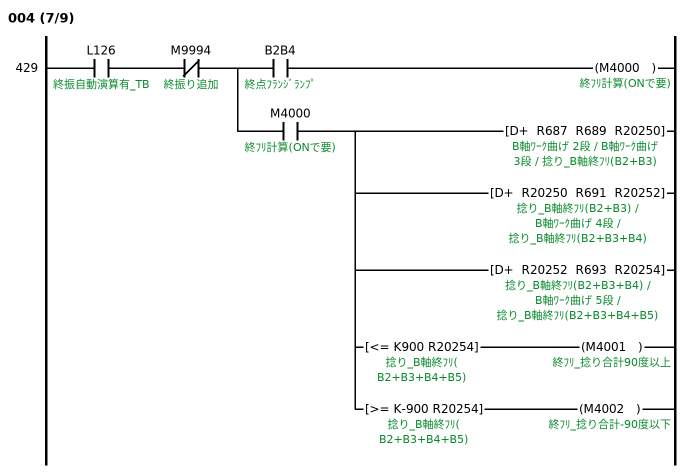
429   LD      L126  ; 終振自動演算有_TB
      ANI     M9994  ; 終振り追加
      MPS
      AND     B2B4  ; 終点ﾌﾗﾝｼﾞﾗﾝﾌﾟ
      OUT     M4000  ; 終ﾌﾘ計算(ONで要)
      MPP
      AND     M4000  ; 終ﾌﾘ計算(ONで要)
      D+      R687 R689 R20250  ; B軸ﾜｰｸ曲げ 2段 / B軸ﾜｰｸ曲げ 3段 / 捻り_B軸終ﾌﾘ(B2+B3)
      D+      R20250 R691 R20252  ; B軸ﾜｰｸ曲げ 4段 / 捻り_B軸終ﾌﾘ(B2+B3+B4)
      D+      R20252 R693 R20254  ; B軸ﾜｰｸ曲げ 5段 / 捻り_B軸終ﾌﾘ(B2+B3+B4+B5)
      MPS
      AND<=   K900 R20254  ; 捻り_B軸終ﾌﾘ(B2+B3+B4+B5)
      OUT     M4001  ; 終ﾌﾘ_捻り合計90度以上
      MPP
      AND>=   K-900 R20254  ; 捻り_B軸終ﾌﾘ(B2+B3+B4+B5)
      OUT     M4002  ; 終ﾌﾘ_捻り合計-90度以下
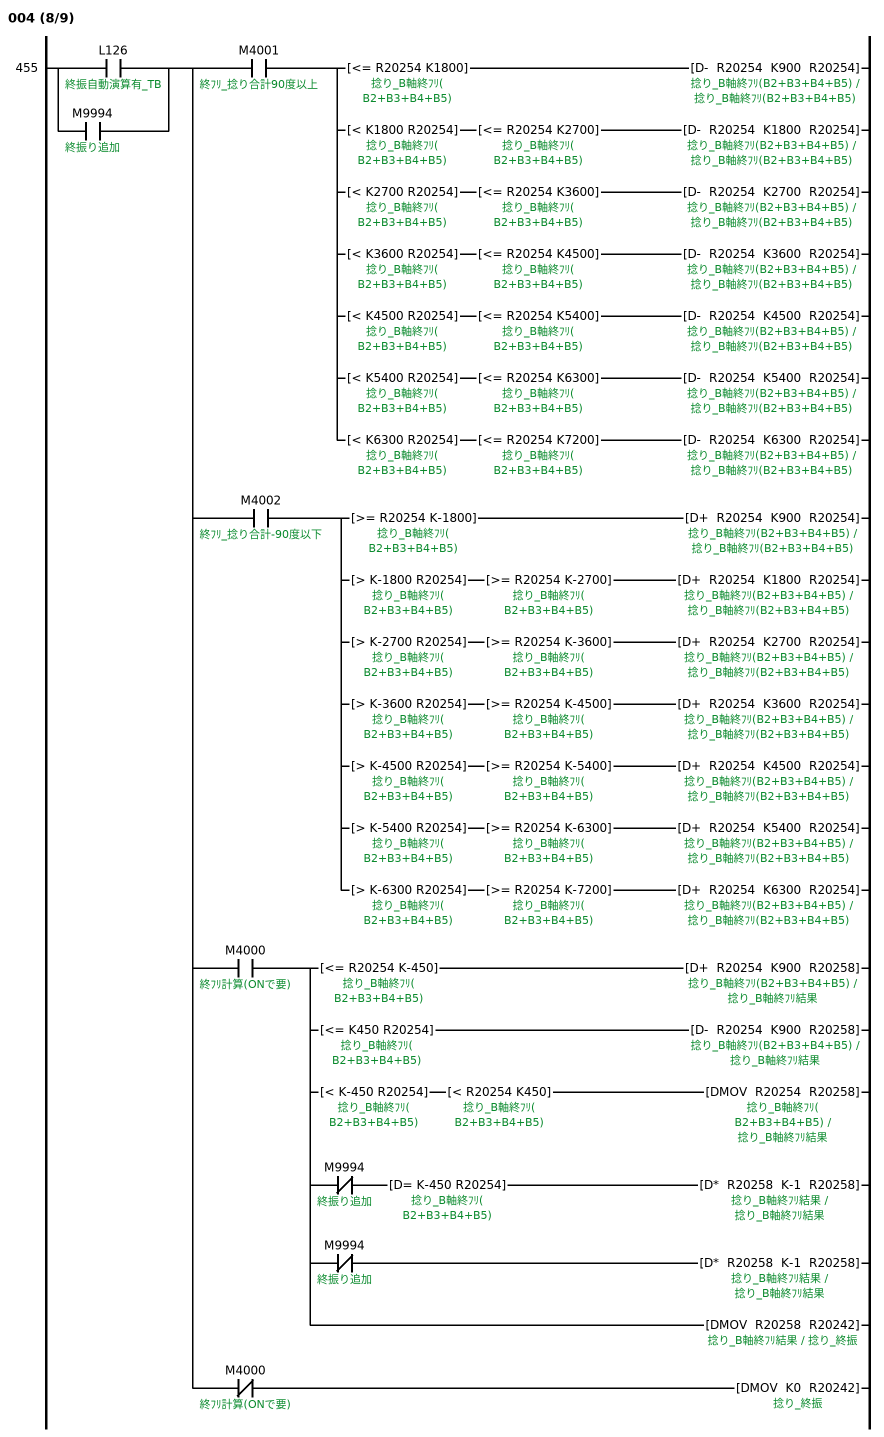
455   LD      L126  ; 終振自動演算有_TB
      OR      M9994  ; 終振り追加
      MPS
      AND     M4001  ; 終ﾌﾘ_捻り合計90度以上
      MPS
      AND<=   R20254 K1800  ; 捻り_B軸終ﾌﾘ(B2+B3+B4+B5)
      D-      R20254 K900 R20254
      MRD
      AND<    K1800 R20254  ; 捻り_B軸終ﾌﾘ(B2+B3+B4+B5)
      AND<=   R20254 K2700  ; 捻り_B軸終ﾌﾘ(B2+B3+B4+B5)
      D-      R20254 K1800 R20254
      MRD
      AND<    K2700 R20254  ; 捻り_B軸終ﾌﾘ(B2+B3+B4+B5)
      AND<=   R20254 K3600  ; 捻り_B軸終ﾌﾘ(B2+B3+B4+B5)
      D-      R20254 K2700 R20254
      MRD
      AND<    K3600 R20254  ; 捻り_B軸終ﾌﾘ(B2+B3+B4+B5)
      AND<=   R20254 K4500  ; 捻り_B軸終ﾌﾘ(B2+B3+B4+B5)
      D-      R20254 K3600 R20254
      MRD
      AND<    K4500 R20254  ; 捻り_B軸終ﾌﾘ(B2+B3+B4+B5)
      AND<=   R20254 K5400  ; 捻り_B軸終ﾌﾘ(B2+B3+B4+B5)
      D-      R20254 K4500 R20254
      MRD
      AND<    K5400 R20254  ; 捻り_B軸終ﾌﾘ(B2+B3+B4+B5)
      AND<=   R20254 K6300  ; 捻り_B軸終ﾌﾘ(B2+B3+B4+B5)
      D-      R20254 K5400 R20254
      MPP
      AND<    K6300 R20254  ; 捻り_B軸終ﾌﾘ(B2+B3+B4+B5)
      AND<=   R20254 K7200  ; 捻り_B軸終ﾌﾘ(B2+B3+B4+B5)
      D-      R20254 K6300 R20254
      MRD
      AND     M4002  ; 終ﾌﾘ_捻り合計-90度以下
      MPS
      AND>=   R20254 K-1800  ; 捻り_B軸終ﾌﾘ(B2+B3+B4+B5)
      D+      R20254 K900 R20254
      MRD
      AND>    K-1800 R20254  ; 捻り_B軸終ﾌﾘ(B2+B3+B4+B5)
      AND>=   R20254 K-2700  ; 捻り_B軸終ﾌﾘ(B2+B3+B4+B5)
      D+      R20254 K1800 R20254
      MRD
      AND>    K-2700 R20254  ; 捻り_B軸終ﾌﾘ(B2+B3+B4+B5)
      AND>=   R20254 K-3600  ; 捻り_B軸終ﾌﾘ(B2+B3+B4+B5)
      D+      R20254 K2700 R20254
      MRD
      AND>    K-3600 R20254  ; 捻り_B軸終ﾌﾘ(B2+B3+B4+B5)
      AND>=   R20254 K-4500  ; 捻り_B軸終ﾌﾘ(B2+B3+B4+B5)
      D+      R20254 K3600 R20254
      MRD
      AND>    K-4500 R20254  ; 捻り_B軸終ﾌﾘ(B2+B3+B4+B5)
      AND>=   R20254 K-5400  ; 捻り_B軸終ﾌﾘ(B2+B3+B4+B5)
      D+      R20254 K4500 R20254
      MRD
      AND>    K-5400 R20254  ; 捻り_B軸終ﾌﾘ(B2+B3+B4+B5)
      AND>=   R20254 K-6300  ; 捻り_B軸終ﾌﾘ(B2+B3+B4+B5)
      D+      R20254 K5400 R20254
      MPP
      AND>    K-6300 R20254  ; 捻り_B軸終ﾌﾘ(B2+B3+B4+B5)
      AND>=   R20254 K-7200  ; 捻り_B軸終ﾌﾘ(B2+B3+B4+B5)
      D+      R20254 K6300 R20254
      MRD
      AND     M4000  ; 終ﾌﾘ計算(ONで要)
      MPS
      AND<=   R20254 K-450  ; 捻り_B軸終ﾌﾘ(B2+B3+B4+B5)
      D+      R20254 K900 R20258  ; 捻り_B軸終ﾌﾘ結果
      MRD
      AND<=   K450 R20254  ; 捻り_B軸終ﾌﾘ(B2+B3+B4+B5)
      D-      R20254 K900 R20258
      MRD
      AND<    K-450 R20254  ; 捻り_B軸終ﾌﾘ(B2+B3+B4+B5)
      AND<    R20254 K450  ; 捻り_B軸終ﾌﾘ(B2+B3+B4+B5)
      DMOV    R20254 R20258
      MRD
      ANI     M9994  ; 終振り追加
      ANDD=   K-450 R20254  ; 捻り_B軸終ﾌﾘ(B2+B3+B4+B5)
      D*      R20258 K-1 R20258
      MRD
      ANI     M9994  ; 終振り追加
      D*      R20258 K-1 R20258
      MPP
      DMOV    R20258 R20242
      MPP
      ANI     M4000  ; 終ﾌﾘ計算(ONで要)
      DMOV    K0 R20242
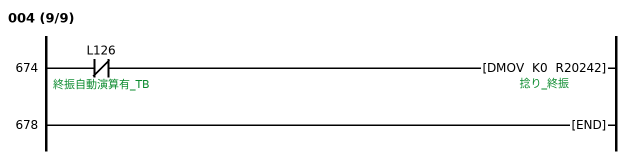
674   LDI     L126  ; 終振自動演算有_TB
      DMOV    K0 R20242
678   END
END_PROGRAM

PROGRAM 006  // 原点復帰
; 
      P600
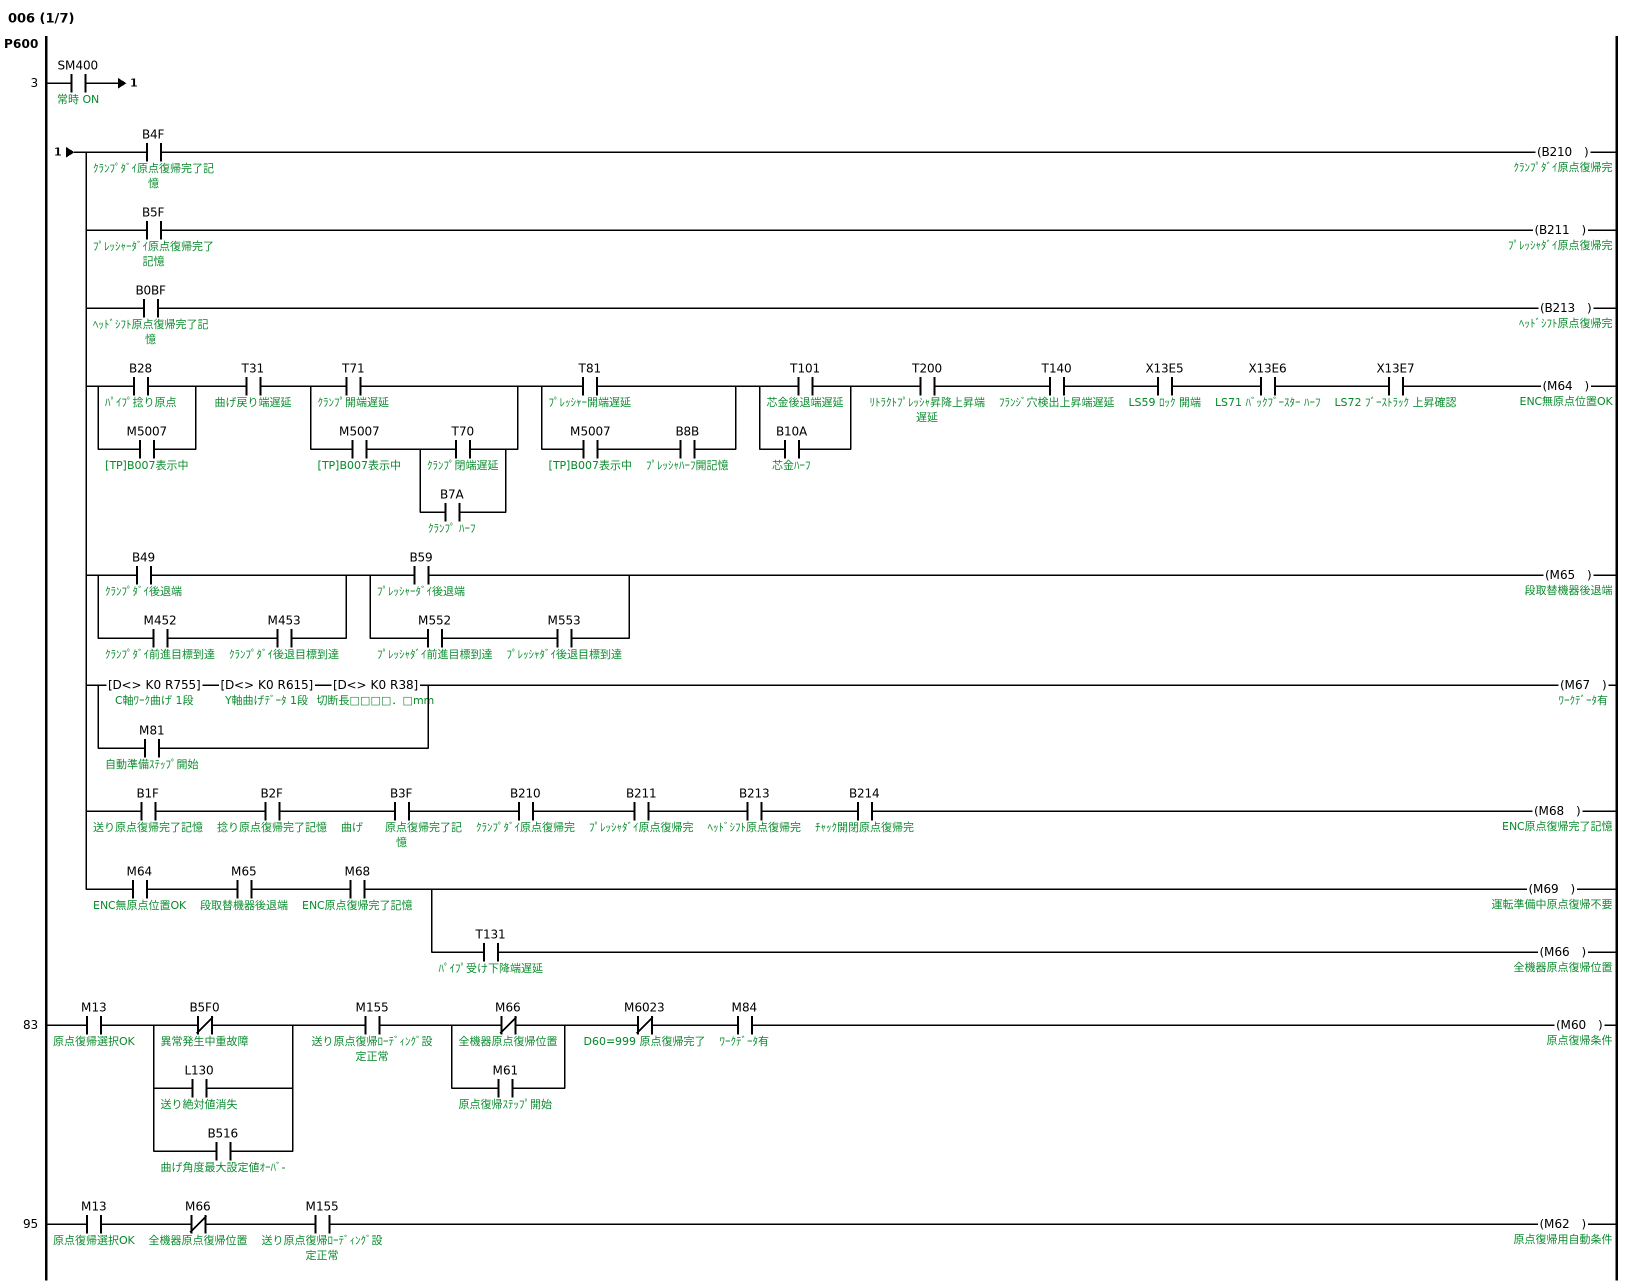
3     LD      SM400  ; 常時 ON
      MPS
      AND     B4F  ; ｸﾗﾝﾌﾟﾀﾞｲ原点復帰完了記憶
      OUT     B210  ; ｸﾗﾝﾌﾟﾀﾞｲ原点復帰完
      MRD
      AND     B5F  ; ﾌﾟﾚｯｼｬｰﾀﾞｲ原点復帰完了記憶
      OUT     B211  ; ﾌﾟﾚｯｼｬﾀﾞｲ原点復帰完
      MRD
      AND     B0BF  ; ﾍｯﾄﾞｼﾌﾄ原点復帰完了記憶
      OUT     B213  ; ﾍｯﾄﾞｼﾌﾄ原点復帰完
      MRD
      LD      B28  ; ﾊﾟｲﾌﾟ捻り原点
      OR      M5007  ; [TP]B007表示中
      ANB
      AND     T31  ; 曲げ戻り端遅延
      LD      T71  ; ｸﾗﾝﾌﾟ開端遅延
      LD      M5007  ; [TP]B007表示中
      LD      T70  ; ｸﾗﾝﾌﾟ閉端遅延
      OR      B7A  ; ｸﾗﾝﾌﾟ ﾊｰﾌ
      ANB
      ORB
      ANB
      LD      T81  ; ﾌﾟﾚｯｼｬｰ開端遅延
      LD      M5007  ; [TP]B007表示中
      AND     B8B  ; ﾌﾟﾚｯｼｬﾊｰﾌ開記憶
      ORB
      ANB
      LD      T101  ; 芯金後退端遅延
      OR      B10A  ; 芯金ﾊｰﾌ
      ANB
      AND     T200  ; ﾘﾄﾗｸﾄﾌﾟﾚｯｼｬ昇降上昇端遅延
      AND     T140  ; ﾌﾗﾝｼﾞ穴検出上昇端遅延
      AND     X13E5  ; LS59 ﾛｯｸ 開端
      AND     X13E6  ; LS71 ﾊﾞｯｸﾌﾞｰｽﾀｰ ﾊｰﾌ
      AND     X13E7  ; LS72 ﾌﾞｰｽﾄﾗｯｸ 上昇確認
      OUT     M64  ; ENC無原点位置OK
      MRD
      LD      B49  ; ｸﾗﾝﾌﾟﾀﾞｲ後退端
      LD      M452  ; ｸﾗﾝﾌﾟﾀﾞｲ前進目標到達
      AND     M453  ; ｸﾗﾝﾌﾟﾀﾞｲ後退目標到達
      ORB
      ANB
      LD      B59  ; ﾌﾟﾚｯｼｬｰﾀﾞｲ後退端
      LD      M552  ; ﾌﾟﾚｯｼｬﾀﾞｲ前進目標到達
      AND     M553  ; ﾌﾟﾚｯｼｬﾀﾞｲ後退目標到達
      ORB
      ANB
      OUT     M65  ; 段取替機器後退端
      MRD
      LDD<>   K0 R755  ; C軸ﾜｰｸ曲げ 1段
      ANDD<>  K0 R615  ; Y軸曲げﾃﾞｰﾀ 1段
      ANDD<>  K0 R38  ; 切断長□□□□．□mm
      OR      M81  ; 自動準備ｽﾃｯﾌﾟ開始
      ANB
      OUT     M67  ; ﾜｰｸﾃﾞｰﾀ有
      MRD
      AND     B1F  ; 送り原点復帰完了記憶
      AND     B2F  ; 捻り原点復帰完了記憶
      AND     B3F  ; 曲げ　　原点復帰完了記憶
      AND     B210  ; ｸﾗﾝﾌﾟﾀﾞｲ原点復帰完
      AND     B211  ; ﾌﾟﾚｯｼｬﾀﾞｲ原点復帰完
      AND     B213  ; ﾍｯﾄﾞｼﾌﾄ原点復帰完
      AND     B214  ; ﾁｬｯｸ開閉原点復帰完
      OUT     M68  ; ENC原点復帰完了記憶
      MPP
      AND     M64  ; ENC無原点位置OK
      AND     M65  ; 段取替機器後退端
      AND     M68  ; ENC原点復帰完了記憶
      OUT     M69  ; 運転準備中原点復帰不要
      AND     T131  ; ﾊﾟｲﾌﾟ受け下降端遅延
      OUT     M66  ; 全機器原点復帰位置
83    LD      M13  ; 原点復帰選択OK
      LDI     B5F0  ; 異常発生中重故障
      OR      L130  ; 送り絶対値消失
      OR      B516  ; 曲げ角度最大設定値ｵｰﾊﾞ-
      ANB
      AND     M155  ; 送り原点復帰ﾛｰﾃﾞｨﾝｸﾞ設定正常
      LDI     M66  ; 全機器原点復帰位置
      OR      M61  ; 原点復帰ｽﾃｯﾌﾟ開始
      ANB
      ANI     M6023  ; D60=999 原点復帰完了
      AND     M84  ; ﾜｰｸﾃﾞｰﾀ有
      OUT     M60  ; 原点復帰条件
95    LD      M13  ; 原点復帰選択OK
      ANI     M66  ; 全機器原点復帰位置
      AND     M155  ; 送り原点復帰ﾛｰﾃﾞｨﾝｸﾞ設定正常
      OUT     M62  ; 原点復帰用自動条件
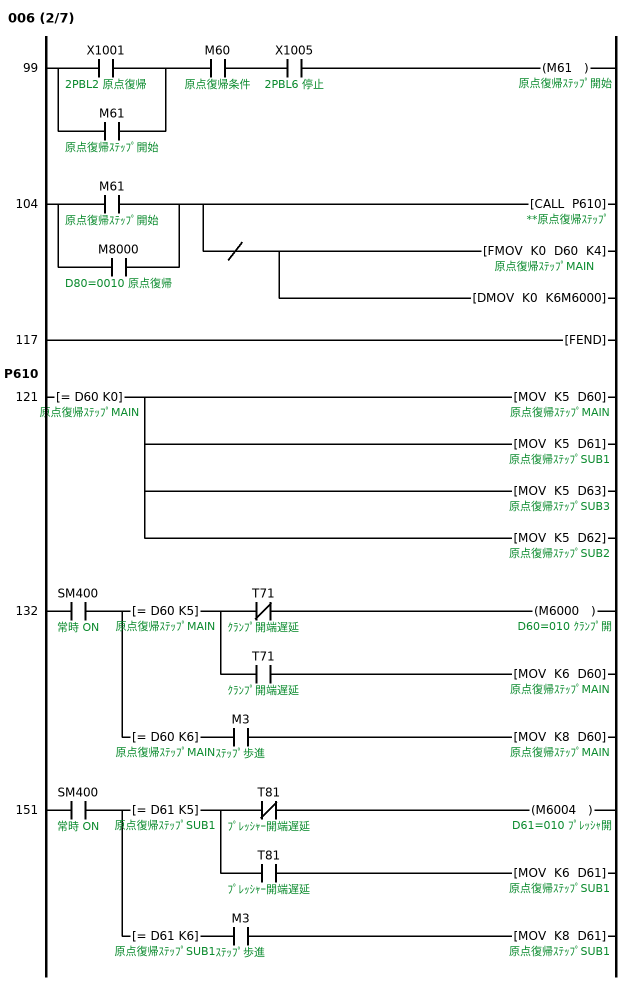
99    LD      X1001  ; 2PBL2 原点復帰
      OR      M61  ; 原点復帰ｽﾃｯﾌﾟ開始
      AND     M60  ; 原点復帰条件
      AND     X1005  ; 2PBL6 停止
      OUT     M61  ; 原点復帰ｽﾃｯﾌﾟ開始
104   LD      M61  ; 原点復帰ｽﾃｯﾌﾟ開始
      OR      M8000  ; D80=0010 原点復帰
      CALL    P610  ; **原点復帰ｽﾃｯﾌﾟ
      INV
      FMOV    K0 D60 K4  ; 原点復帰ｽﾃｯﾌﾟMAIN
      DMOV    K0 K6M6000  ; D60=010 ｸﾗﾝﾌﾟ開
117   FEND
; 
      P610
121   LD=     D60 K0  ; 原点復帰ｽﾃｯﾌﾟMAIN
      MOV     K5 D60
      MOV     K5 D61  ; 原点復帰ｽﾃｯﾌﾟSUB1
      MOV     K5 D63  ; 原点復帰ｽﾃｯﾌﾟSUB3
      MOV     K5 D62  ; 原点復帰ｽﾃｯﾌﾟSUB2
132   LD      SM400  ; 常時 ON
      MPS
      AND=    D60 K5  ; 原点復帰ｽﾃｯﾌﾟMAIN
      MPS
      ANI     T71  ; ｸﾗﾝﾌﾟ開端遅延
      OUT     M6000  ; D60=010 ｸﾗﾝﾌﾟ開
      MPP
      AND     T71  ; ｸﾗﾝﾌﾟ開端遅延
      MOV     K6 D60
      MPP
      AND=    D60 K6  ; 原点復帰ｽﾃｯﾌﾟMAIN
      AND     M3  ; ｽﾃｯﾌﾟ歩進
      MOV     K8 D60
151   LD      SM400  ; 常時 ON
      MPS
      AND=    D61 K5  ; 原点復帰ｽﾃｯﾌﾟSUB1
      MPS
      ANI     T81  ; ﾌﾟﾚｯｼｬｰ開端遅延
      OUT     M6004  ; D61=010 ﾌﾟﾚｯｼｬ開
      MPP
      AND     T81  ; ﾌﾟﾚｯｼｬｰ開端遅延
      MOV     K6 D61
      MPP
      AND=    D61 K6  ; 原点復帰ｽﾃｯﾌﾟSUB1
      AND     M3  ; ｽﾃｯﾌﾟ歩進
      MOV     K8 D61
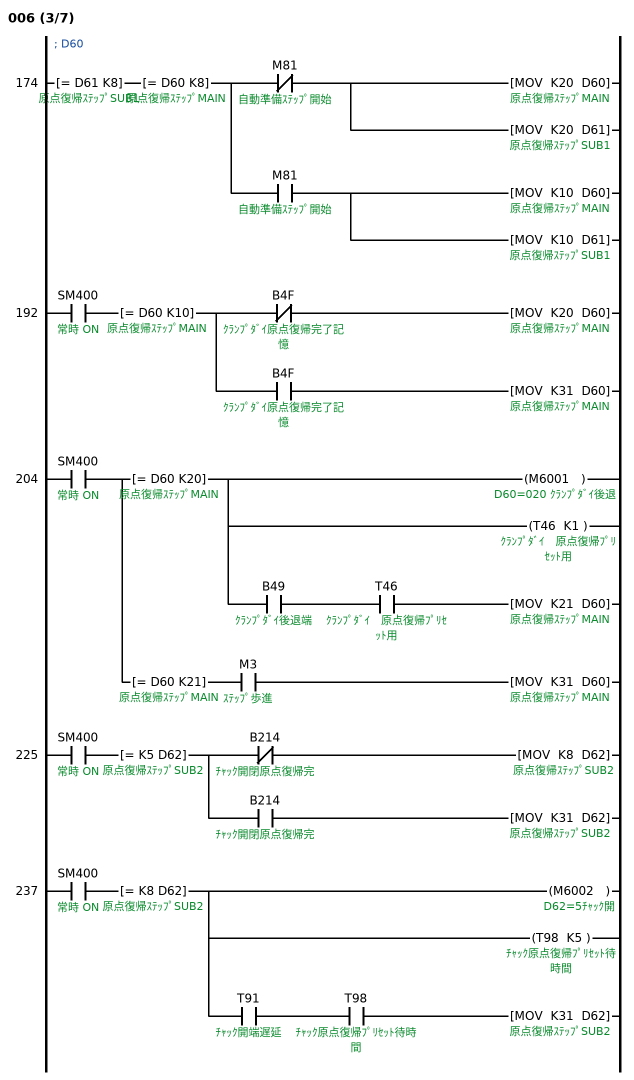
; D60
174   LD=     D61 K8  ; 原点復帰ｽﾃｯﾌﾟSUB1
      AND=    D60 K8  ; 原点復帰ｽﾃｯﾌﾟMAIN
      MPS
      ANI     M81  ; 自動準備ｽﾃｯﾌﾟ開始
      MOV     K20 D60
      MOV     K20 D61
      MPP
      AND     M81  ; 自動準備ｽﾃｯﾌﾟ開始
      MOV     K10 D60
      MOV     K10 D61
192   LD      SM400  ; 常時 ON
      AND=    D60 K10  ; 原点復帰ｽﾃｯﾌﾟMAIN
      MPS
      ANI     B4F  ; ｸﾗﾝﾌﾟﾀﾞｲ原点復帰完了記憶
      MOV     K20 D60
      MPP
      AND     B4F  ; ｸﾗﾝﾌﾟﾀﾞｲ原点復帰完了記憶
      MOV     K31 D60
204   LD      SM400  ; 常時 ON
      MPS
      AND=    D60 K20  ; 原点復帰ｽﾃｯﾌﾟMAIN
      OUT     M6001  ; D60=020 ｸﾗﾝﾌﾟﾀﾞｲ後退
      OUT     T46 K1  ; ｸﾗﾝﾌﾟﾀﾞｲ　原点復帰ﾌﾟﾘｾｯﾄ用
      AND     B49  ; ｸﾗﾝﾌﾟﾀﾞｲ後退端
      AND     T46  ; ｸﾗﾝﾌﾟﾀﾞｲ　原点復帰ﾌﾟﾘｾｯﾄ用
      MOV     K21 D60
      MPP
      AND=    D60 K21  ; 原点復帰ｽﾃｯﾌﾟMAIN
      AND     M3  ; ｽﾃｯﾌﾟ歩進
      MOV     K31 D60
225   LD      SM400  ; 常時 ON
      AND=    K5 D62  ; 原点復帰ｽﾃｯﾌﾟSUB2
      MPS
      ANI     B214  ; ﾁｬｯｸ開閉原点復帰完
      MOV     K8 D62
      MPP
      AND     B214  ; ﾁｬｯｸ開閉原点復帰完
      MOV     K31 D62
237   LD      SM400  ; 常時 ON
      AND=    K8 D62  ; 原点復帰ｽﾃｯﾌﾟSUB2
      OUT     M6002  ; D62=5ﾁｬｯｸ開
      OUT     T98 K5  ; ﾁｬｯｸ原点復帰ﾌﾟﾘｾｯﾄ待時間
      AND     T91  ; ﾁｬｯｸ開端遅延
      AND     T98  ; ﾁｬｯｸ原点復帰ﾌﾟﾘｾｯﾄ待時間
      MOV     K31 D62
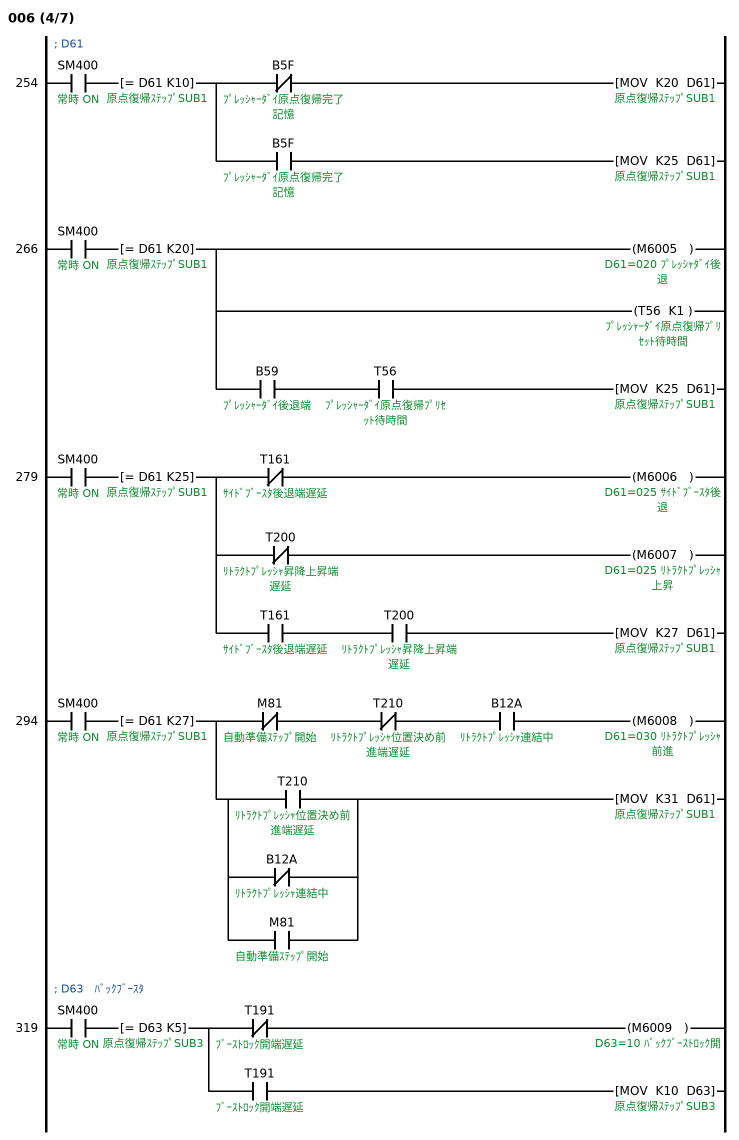
; D61
254   LD      SM400  ; 常時 ON
      AND=    D61 K10  ; 原点復帰ｽﾃｯﾌﾟSUB1
      MPS
      ANI     B5F  ; ﾌﾟﾚｯｼｬｰﾀﾞｲ原点復帰完了記憶
      MOV     K20 D61
      MPP
      AND     B5F  ; ﾌﾟﾚｯｼｬｰﾀﾞｲ原点復帰完了記憶
      MOV     K25 D61
266   LD      SM400  ; 常時 ON
      AND=    D61 K20  ; 原点復帰ｽﾃｯﾌﾟSUB1
      OUT     M6005  ; D61=020 ﾌﾟﾚｯｼｬﾀﾞｲ後退
      OUT     T56 K1  ; ﾌﾟﾚｯｼｬｰﾀﾞｲ原点復帰ﾌﾟﾘｾｯﾄ待時間
      AND     B59  ; ﾌﾟﾚｯｼｬｰﾀﾞｲ後退端
      AND     T56  ; ﾌﾟﾚｯｼｬｰﾀﾞｲ原点復帰ﾌﾟﾘｾｯﾄ待時間
      MOV     K25 D61
279   LD      SM400  ; 常時 ON
      AND=    D61 K25  ; 原点復帰ｽﾃｯﾌﾟSUB1
      MPS
      ANI     T161  ; ｻｲﾄﾞﾌﾞｰｽﾀ後退端遅延
      OUT     M6006  ; D61=025 ｻｲﾄﾞﾌﾞｰｽﾀ後退
      MRD
      ANI     T200  ; ﾘﾄﾗｸﾄﾌﾟﾚｯｼｬ昇降上昇端遅延
      OUT     M6007  ; D61=025 ﾘﾄﾗｸﾄﾌﾟﾚｯｼｬ上昇
      MPP
      AND     T161  ; ｻｲﾄﾞﾌﾞｰｽﾀ後退端遅延
      AND     T200  ; ﾘﾄﾗｸﾄﾌﾟﾚｯｼｬ昇降上昇端遅延
      MOV     K27 D61
294   LD      SM400  ; 常時 ON
      AND=    D61 K27  ; 原点復帰ｽﾃｯﾌﾟSUB1
      MPS
      ANI     M81  ; 自動準備ｽﾃｯﾌﾟ開始
      ANI     T210  ; ﾘﾄﾗｸﾄﾌﾟﾚｯｼｬ位置決め前進端遅延
      AND     B12A  ; ﾘﾄﾗｸﾄﾌﾟﾚｯｼｬ連結中
      OUT     M6008  ; D61=030 ﾘﾄﾗｸﾄﾌﾟﾚｯｼｬ前進
      MPP
      LD      T210  ; ﾘﾄﾗｸﾄﾌﾟﾚｯｼｬ位置決め前進端遅延
      ORI     B12A  ; ﾘﾄﾗｸﾄﾌﾟﾚｯｼｬ連結中
      OR      M81  ; 自動準備ｽﾃｯﾌﾟ開始
      ANB
      MOV     K31 D61
; D63　ﾊﾞｯｸﾌﾞｰｽﾀ
319   LD      SM400  ; 常時 ON
      AND=    D63 K5  ; 原点復帰ｽﾃｯﾌﾟSUB3
      MPS
      ANI     T191  ; ﾌﾞｰｽﾄﾛｯｸ開端遅延
      OUT     M6009  ; D63=10 ﾊﾞｯｸﾌﾞｰｽﾄﾛｯｸ開
      MPP
      AND     T191  ; ﾌﾞｰｽﾄﾛｯｸ開端遅延
      MOV     K10 D63
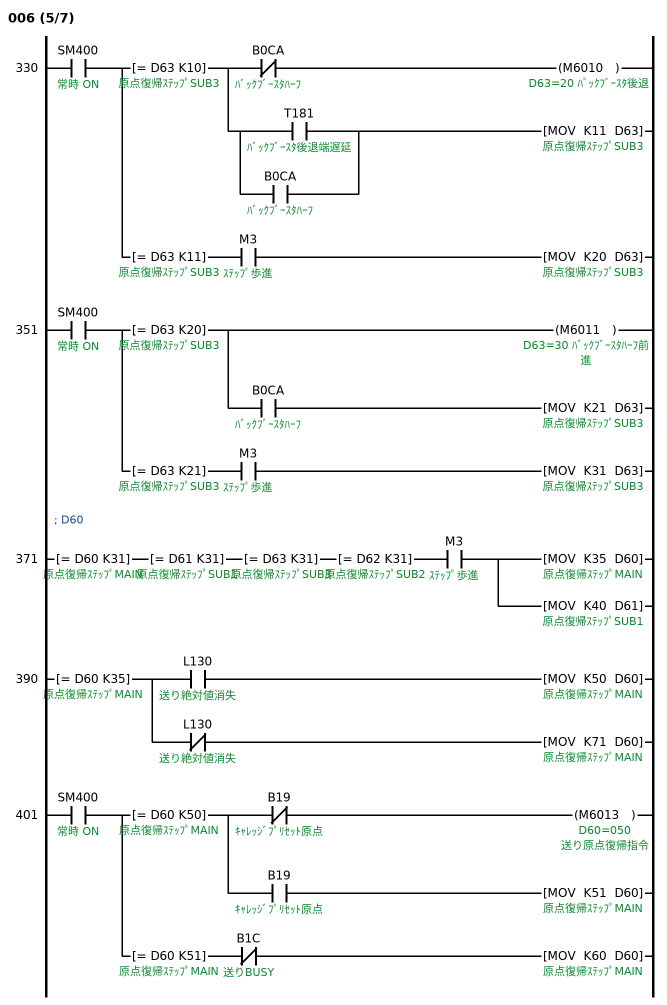
330   LD      SM400  ; 常時 ON
      MPS
      AND=    D63 K10  ; 原点復帰ｽﾃｯﾌﾟSUB3
      MPS
      ANI     B0CA  ; ﾊﾞｯｸﾌﾞｰｽﾀﾊｰﾌ
      OUT     M6010  ; D63=20 ﾊﾞｯｸﾌﾞｰｽﾀ後退
      MPP
      LD      T181  ; ﾊﾞｯｸﾌﾞｰｽﾀ後退端遅延
      OR      B0CA  ; ﾊﾞｯｸﾌﾞｰｽﾀﾊｰﾌ
      ANB
      MOV     K11 D63
      MPP
      AND=    D63 K11  ; 原点復帰ｽﾃｯﾌﾟSUB3
      AND     M3  ; ｽﾃｯﾌﾟ歩進
      MOV     K20 D63
351   LD      SM400  ; 常時 ON
      MPS
      AND=    D63 K20  ; 原点復帰ｽﾃｯﾌﾟSUB3
      OUT     M6011  ; D63=30 ﾊﾞｯｸﾌﾞｰｽﾀﾊｰﾌ前進
      AND     B0CA  ; ﾊﾞｯｸﾌﾞｰｽﾀﾊｰﾌ
      MOV     K21 D63
      MPP
      AND=    D63 K21  ; 原点復帰ｽﾃｯﾌﾟSUB3
      AND     M3  ; ｽﾃｯﾌﾟ歩進
      MOV     K31 D63
; D60
371   LD=     D60 K31  ; 原点復帰ｽﾃｯﾌﾟMAIN
      AND=    D61 K31  ; 原点復帰ｽﾃｯﾌﾟSUB1
      AND=    D63 K31  ; 原点復帰ｽﾃｯﾌﾟSUB3
      AND=    D62 K31  ; 原点復帰ｽﾃｯﾌﾟSUB2
      AND     M3  ; ｽﾃｯﾌﾟ歩進
      MOV     K35 D60
      MOV     K40 D61
; 
390   LD=     D60 K35  ; 原点復帰ｽﾃｯﾌﾟMAIN
      MPS
      AND     L130  ; 送り絶対値消失
      MOV     K50 D60
      MPP
      ANI     L130  ; 送り絶対値消失
      MOV     K71 D60
401   LD      SM400  ; 常時 ON
      MPS
      AND=    D60 K50  ; 原点復帰ｽﾃｯﾌﾟMAIN
      MPS
      ANI     B19  ; ｷｬﾚｯｼﾞﾌﾟﾘｾｯﾄ原点
      OUT     M6013  ; D60=050 送り原点復帰指令
      MPP
      AND     B19  ; ｷｬﾚｯｼﾞﾌﾟﾘｾｯﾄ原点
      MOV     K51 D60
      MPP
      AND=    D60 K51  ; 原点復帰ｽﾃｯﾌﾟMAIN
      ANI     B1C  ; 送りBUSY
      MOV     K60 D60
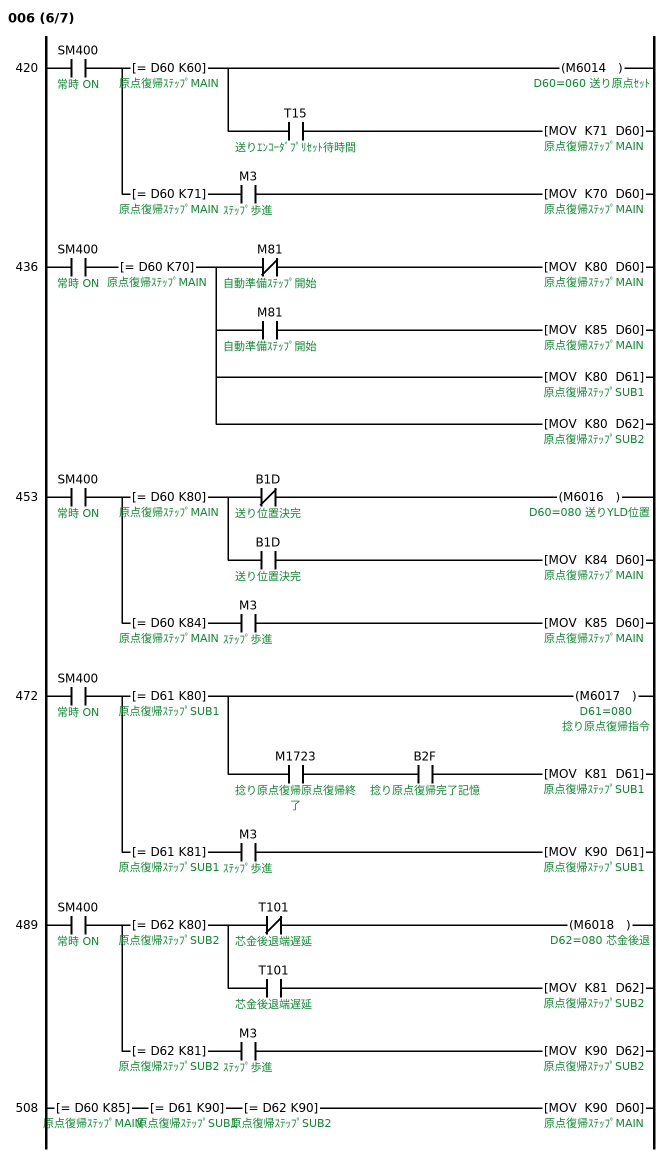
420   LD      SM400  ; 常時 ON
      MPS
      AND=    D60 K60  ; 原点復帰ｽﾃｯﾌﾟMAIN
      OUT     M6014  ; D60=060 送り原点ｾｯﾄ
      AND     T15  ; 送りｴﾝｺｰﾀﾞﾌﾟﾘｾｯﾄ待時間
      MOV     K71 D60
      MPP
      AND=    D60 K71  ; 原点復帰ｽﾃｯﾌﾟMAIN
      AND     M3  ; ｽﾃｯﾌﾟ歩進
      MOV     K70 D60
436   LD      SM400  ; 常時 ON
      AND=    D60 K70  ; 原点復帰ｽﾃｯﾌﾟMAIN
      MPS
      ANI     M81  ; 自動準備ｽﾃｯﾌﾟ開始
      MOV     K80 D60
      MRD
      AND     M81  ; 自動準備ｽﾃｯﾌﾟ開始
      MOV     K85 D60
      MPP
      MOV     K80 D61
      MOV     K80 D62
453   LD      SM400  ; 常時 ON
      MPS
      AND=    D60 K80  ; 原点復帰ｽﾃｯﾌﾟMAIN
      MPS
      ANI     B1D  ; 送り位置決完
      OUT     M6016  ; D60=080 送りYLD位置
      MPP
      AND     B1D  ; 送り位置決完
      MOV     K84 D60
      MPP
      AND=    D60 K84  ; 原点復帰ｽﾃｯﾌﾟMAIN
      AND     M3  ; ｽﾃｯﾌﾟ歩進
      MOV     K85 D60
472   LD      SM400  ; 常時 ON
      MPS
      AND=    D61 K80  ; 原点復帰ｽﾃｯﾌﾟSUB1
      OUT     M6017  ; D61=080 捻り原点復帰指令
      AND     M1723  ; 捻り原点復帰原点復帰終了
      AND     B2F  ; 捻り原点復帰完了記憶
      MOV     K81 D61
      MPP
      AND=    D61 K81  ; 原点復帰ｽﾃｯﾌﾟSUB1
      AND     M3  ; ｽﾃｯﾌﾟ歩進
      MOV     K90 D61
489   LD      SM400  ; 常時 ON
      MPS
      AND=    D62 K80  ; 原点復帰ｽﾃｯﾌﾟSUB2
      MPS
      ANI     T101  ; 芯金後退端遅延
      OUT     M6018  ; D62=080 芯金後退
      MPP
      AND     T101  ; 芯金後退端遅延
      MOV     K81 D62
      MPP
      AND=    D62 K81  ; 原点復帰ｽﾃｯﾌﾟSUB2
      AND     M3  ; ｽﾃｯﾌﾟ歩進
      MOV     K90 D62
508   LD=     D60 K85  ; 原点復帰ｽﾃｯﾌﾟMAIN
      AND=    D61 K90  ; 原点復帰ｽﾃｯﾌﾟSUB1
      AND=    D62 K90  ; 原点復帰ｽﾃｯﾌﾟSUB2
      MOV     K90 D60
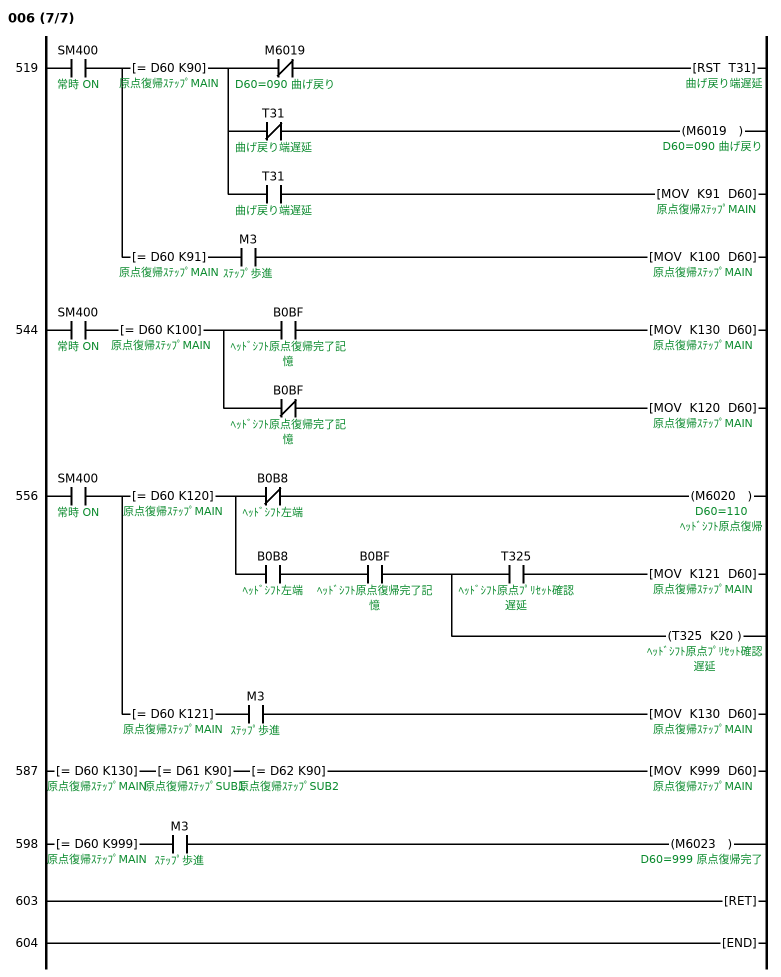
519   LD      SM400  ; 常時 ON
      MPS
      AND=    D60 K90  ; 原点復帰ｽﾃｯﾌﾟMAIN
      MPS
      ANI     M6019  ; D60=090 曲げ戻り
      RST     T31  ; 曲げ戻り端遅延
      MRD
      ANI     T31  ; 曲げ戻り端遅延
      OUT     M6019  ; D60=090 曲げ戻り
      MPP
      AND     T31  ; 曲げ戻り端遅延
      MOV     K91 D60
      MPP
      AND=    D60 K91  ; 原点復帰ｽﾃｯﾌﾟMAIN
      AND     M3  ; ｽﾃｯﾌﾟ歩進
      MOV     K100 D60
544   LD      SM400  ; 常時 ON
      AND=    D60 K100  ; 原点復帰ｽﾃｯﾌﾟMAIN
      MPS
      AND     B0BF  ; ﾍｯﾄﾞｼﾌﾄ原点復帰完了記憶
      MOV     K130 D60
      MPP
      ANI     B0BF  ; ﾍｯﾄﾞｼﾌﾄ原点復帰完了記憶
      MOV     K120 D60
556   LD      SM400  ; 常時 ON
      MPS
      AND=    D60 K120  ; 原点復帰ｽﾃｯﾌﾟMAIN
      MPS
      ANI     B0B8  ; ﾍｯﾄﾞｼﾌﾄ左端
      OUT     M6020  ; D60=110 ﾍｯﾄﾞｼﾌﾄ原点復帰
      MPP
      AND     B0B8  ; ﾍｯﾄﾞｼﾌﾄ左端
      AND     B0BF  ; ﾍｯﾄﾞｼﾌﾄ原点復帰完了記憶
      MPS
      AND     T325  ; ﾍｯﾄﾞｼﾌﾄ原点ﾌﾟﾘｾｯﾄ確認遅延
      MOV     K121 D60
      MPP
      OUT     T325 K20  ; ﾍｯﾄﾞｼﾌﾄ原点ﾌﾟﾘｾｯﾄ確認遅延
      MPP
      AND=    D60 K121  ; 原点復帰ｽﾃｯﾌﾟMAIN
      AND     M3  ; ｽﾃｯﾌﾟ歩進
      MOV     K130 D60
; 
; 
587   LD=     D60 K130  ; 原点復帰ｽﾃｯﾌﾟMAIN
      AND=    D61 K90  ; 原点復帰ｽﾃｯﾌﾟSUB1
      AND=    D62 K90  ; 原点復帰ｽﾃｯﾌﾟSUB2
      MOV     K999 D60
598   LD=     D60 K999  ; 原点復帰ｽﾃｯﾌﾟMAIN
      AND     M3  ; ｽﾃｯﾌﾟ歩進
      OUT     M6023  ; D60=999 原点復帰完了
603   RET
604   END
END_PROGRAM

PROGRAM 007  // 自動
; 
      P700
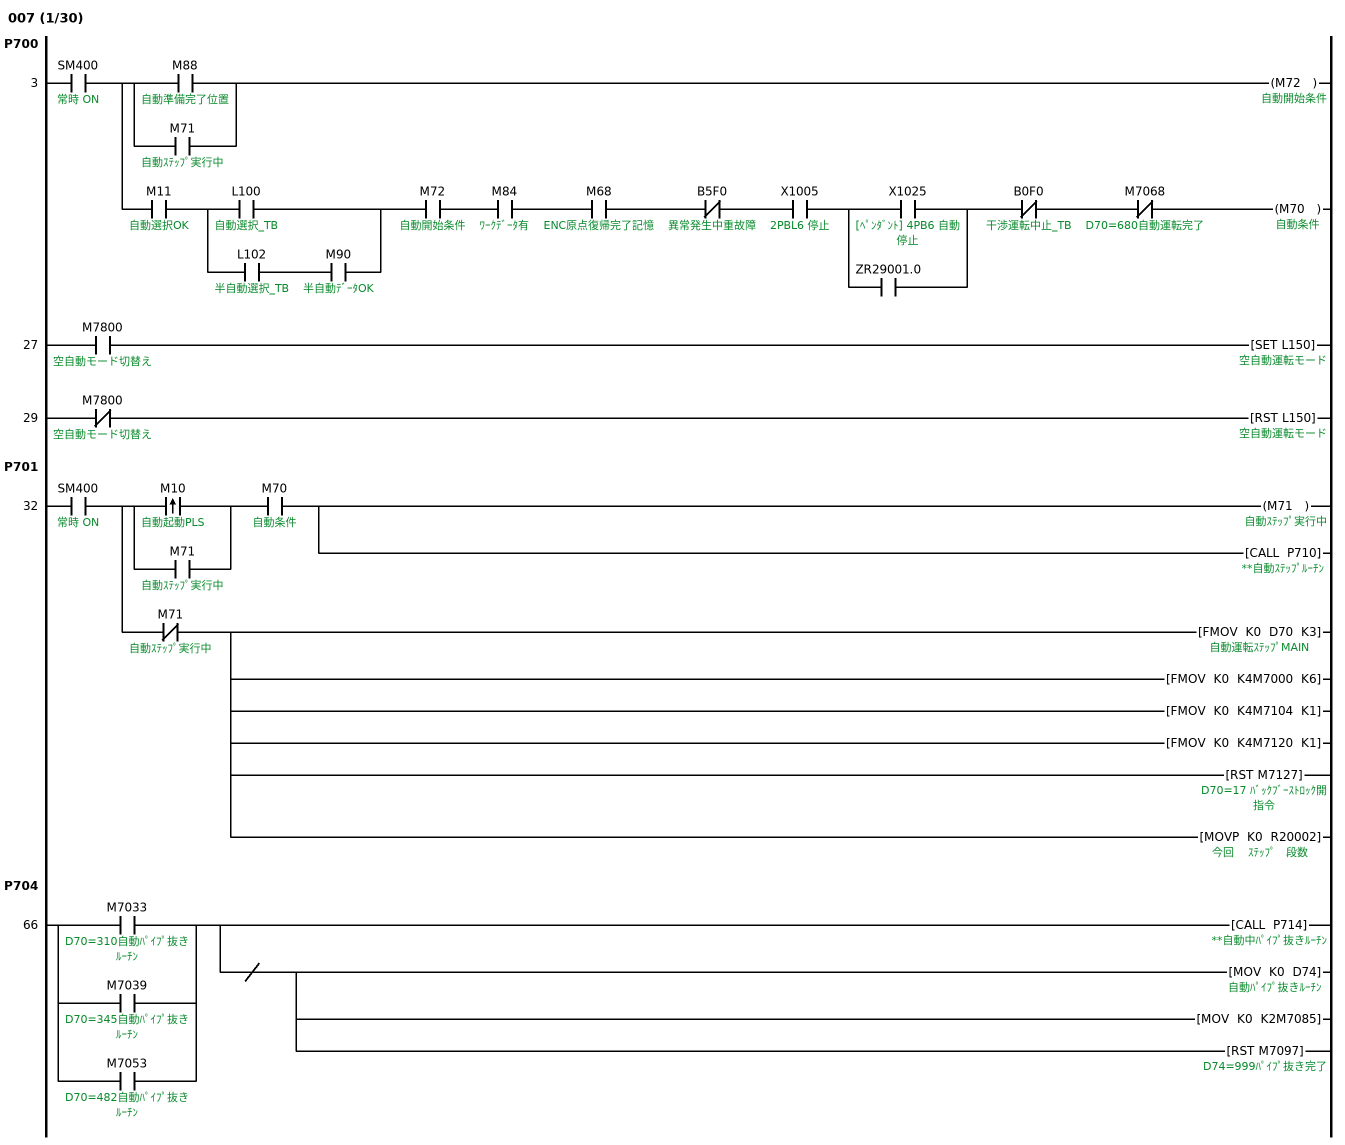
3     LD      SM400  ; 常時 ON
      MPS
      LD      M88  ; 自動準備完了位置
      OR      M71  ; 自動ｽﾃｯﾌﾟ実行中
      ANB
      OUT     M72  ; 自動開始条件
      MPP
      AND     M11  ; 自動選択OK
      LD      L100  ; 自動選択_TB
      LD      L102  ; 半自動選択_TB
      AND     M90  ; 半自動ﾃﾞｰﾀOK
      ORB
      ANB
      AND     M72  ; 自動開始条件
      AND     M84  ; ﾜｰｸﾃﾞｰﾀ有
      AND     M68  ; ENC原点復帰完了記憶
      ANI     B5F0  ; 異常発生中重故障
      AND     X1005  ; 2PBL6 停止
      LD      X1025  ; [ﾍﾟﾝﾀﾞﾝﾄ] 4PB6 自動 停止
      OR      ZR29001.0
      ANB
      ANI     B0F0  ; 干渉運転中止_TB
      ANI     M7068  ; D70=680自動運転完了
      OUT     M70  ; 自動条件
27    LD      M7800  ; 空自動モード切替え
      SET     L150  ; 空自動運転モード
29    LDI     M7800  ; 空自動モード切替え
      RST     L150  ; 空自動運転モード
      P701
32    LD      SM400  ; 常時 ON
      MPS
      LDP     M10  ; 自動起動PLS
      OR      M71  ; 自動ｽﾃｯﾌﾟ実行中
      ANB
      AND     M70  ; 自動条件
      OUT     M71  ; 自動ｽﾃｯﾌﾟ実行中
      CALL    P710  ; **自動ｽﾃｯﾌﾟﾙｰﾁﾝ
      MPP
      ANI     M71  ; 自動ｽﾃｯﾌﾟ実行中
      FMOV    K0 D70 K3  ; 自動運転ｽﾃｯﾌﾟMAIN
      FMOV    K0 K4M7000 K6  ; D70=000ﾃﾞｰﾀ確認
      FMOV    K0 K4M7104 K1  ; D70=590選択ﾛｯﾄ完了
      FMOV    K0 K4M7120 K1  ; D70=307ﾍｯﾄﾞｼﾌﾄ曲げ位置
      RST     M7127  ; D70=17 ﾊﾞｯｸﾌﾞｰｽﾄﾛｯｸ開指令
      MOVP    K0 R20002  ; 今回    ｽﾃｯﾌﾟ   段数
      P704
66    LD      M7033  ; D70=310自動ﾊﾟｲﾌﾟ抜きﾙｰﾁﾝ
      OR      M7039  ; D70=345自動ﾊﾟｲﾌﾟ抜きﾙｰﾁﾝ
      OR      M7053  ; D70=482自動ﾊﾟｲﾌﾟ抜きﾙｰﾁﾝ
      CALL    P714  ; **自動中ﾊﾟｲﾌﾟ抜きﾙｰﾁﾝ
      INV
      MOV     K0 D74  ; 自動ﾊﾟｲﾌﾟ抜きﾙｰﾁﾝ
      MOV     K0 K2M7085  ; D74=000予備
      RST     M7097  ; D74=999ﾊﾟｲﾌﾟ抜き完了
      P705
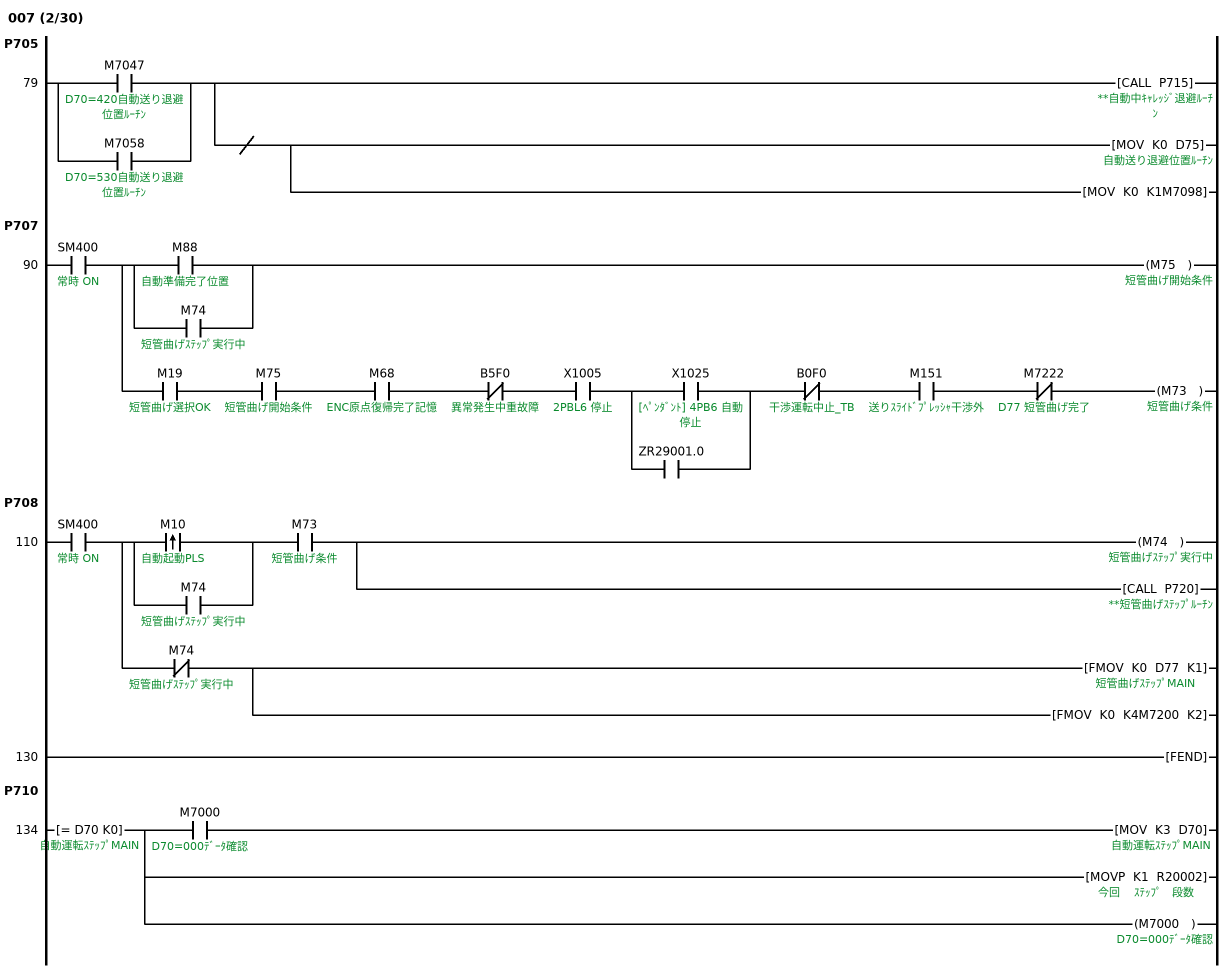
79    LD      M7047  ; D70=420自動送り退避位置ﾙｰﾁﾝ
      OR      M7058  ; D70=530自動送り退避位置ﾙｰﾁﾝ
      CALL    P715  ; **自動中ｷｬﾚｯｼﾞ退避ﾙｰﾁﾝ
      INV
      MOV     K0 D75  ; 自動送り退避位置ﾙｰﾁﾝ
      MOV     K0 K1M7098  ; D75=010送り退避位置
      P707
90    LD      SM400  ; 常時 ON
      MPS
      LD      M88  ; 自動準備完了位置
      OR      M74  ; 短管曲げｽﾃｯﾌﾟ実行中
      ANB
      OUT     M75  ; 短管曲げ開始条件
      MPP
      AND     M19  ; 短管曲げ選択OK
      AND     M75  ; 短管曲げ開始条件
      AND     M68  ; ENC原点復帰完了記憶
      ANI     B5F0  ; 異常発生中重故障
      AND     X1005  ; 2PBL6 停止
      LD      X1025  ; [ﾍﾟﾝﾀﾞﾝﾄ] 4PB6 自動 停止
      OR      ZR29001.0
      ANB
      ANI     B0F0  ; 干渉運転中止_TB
      AND     M151  ; 送りｽﾗｲﾄﾞﾌﾟﾚｯｼｬ干渉外
      ANI     M7222  ; D77 短管曲げ完了
      OUT     M73  ; 短管曲げ条件
      P708
110   LD      SM400  ; 常時 ON
      MPS
      LDP     M10  ; 自動起動PLS
      OR      M74  ; 短管曲げｽﾃｯﾌﾟ実行中
      ANB
      AND     M73  ; 短管曲げ条件
      OUT     M74  ; 短管曲げｽﾃｯﾌﾟ実行中
      CALL    P720  ; **短管曲げｽﾃｯﾌﾟﾙｰﾁﾝ
      MPP
      ANI     M74  ; 短管曲げｽﾃｯﾌﾟ実行中
      FMOV    K0 D77 K1  ; 短管曲げｽﾃｯﾌﾟMAIN
      FMOV    K0 K4M7200 K2
130   FEND
; 
      P710
134   LD=     D70 K0  ; 自動運転ｽﾃｯﾌﾟMAIN
      MPS
      AND     M7000  ; D70=000ﾃﾞｰﾀ確認
      MOV     K3 D70
      MPP
      MOVP    K1 R20002
      OUT     M7000  ; D70=000ﾃﾞｰﾀ確認
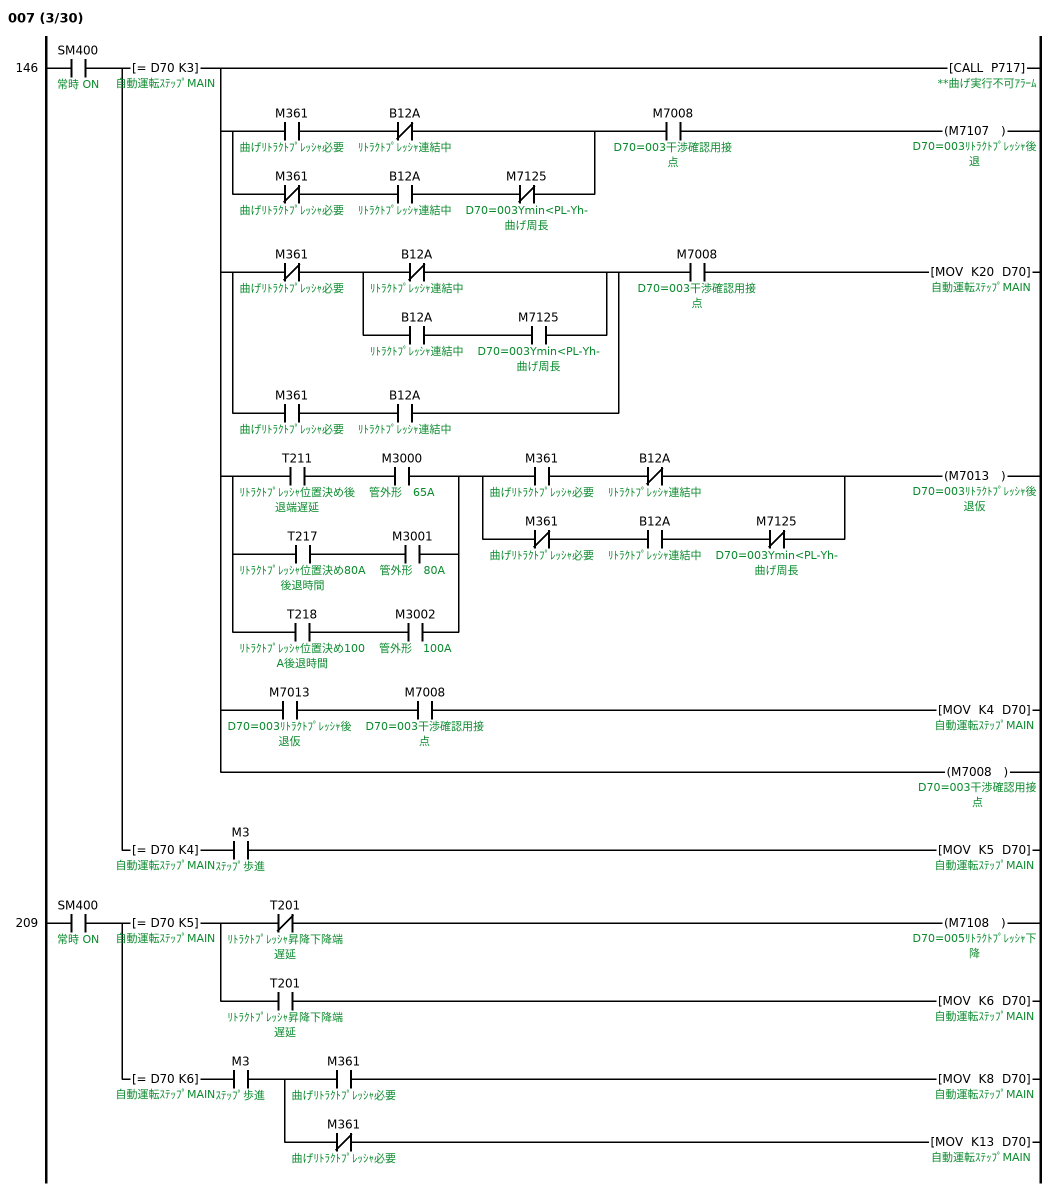
146   LD      SM400  ; 常時 ON
      MPS
      AND=    D70 K3  ; 自動運転ｽﾃｯﾌﾟMAIN
      CALL    P717  ; **曲げ実行不可ｱﾗｰﾑ
      MPS
      LD      M361  ; 曲げﾘﾄﾗｸﾄﾌﾟﾚｯｼｬ必要
      ANI     B12A  ; ﾘﾄﾗｸﾄﾌﾟﾚｯｼｬ連結中
      LDI     M361  ; 曲げﾘﾄﾗｸﾄﾌﾟﾚｯｼｬ必要
      AND     B12A  ; ﾘﾄﾗｸﾄﾌﾟﾚｯｼｬ連結中
      ANI     M7125  ; D70=003Ymin<PL-Yh-曲げ周長
      ORB
      ANB
      AND     M7008  ; D70=003干渉確認用接点
      OUT     M7107  ; D70=003ﾘﾄﾗｸﾄﾌﾟﾚｯｼｬ後退
      MRD
      LDI     M361  ; 曲げﾘﾄﾗｸﾄﾌﾟﾚｯｼｬ必要
      LDI     B12A  ; ﾘﾄﾗｸﾄﾌﾟﾚｯｼｬ連結中
      LD      B12A  ; ﾘﾄﾗｸﾄﾌﾟﾚｯｼｬ連結中
      AND     M7125  ; D70=003Ymin<PL-Yh-曲げ周長
      ORB
      ANB
      LD      M361  ; 曲げﾘﾄﾗｸﾄﾌﾟﾚｯｼｬ必要
      AND     B12A  ; ﾘﾄﾗｸﾄﾌﾟﾚｯｼｬ連結中
      ORB
      ANB
      AND     M7008  ; D70=003干渉確認用接点
      MOV     K20 D70
      MRD
      LD      T211  ; ﾘﾄﾗｸﾄﾌﾟﾚｯｼｬ位置決め後退端遅延
      AND     M3000  ; 管外形　65A
      LD      T217  ; ﾘﾄﾗｸﾄﾌﾟﾚｯｼｬ位置決め80A後退時間
      AND     M3001  ; 管外形　80A
      ORB
      LD      T218  ; ﾘﾄﾗｸﾄﾌﾟﾚｯｼｬ位置決め100A後退時間
      AND     M3002  ; 管外形　100A
      ORB
      ANB
      LD      M361  ; 曲げﾘﾄﾗｸﾄﾌﾟﾚｯｼｬ必要
      ANI     B12A  ; ﾘﾄﾗｸﾄﾌﾟﾚｯｼｬ連結中
      LDI     M361  ; 曲げﾘﾄﾗｸﾄﾌﾟﾚｯｼｬ必要
      AND     B12A  ; ﾘﾄﾗｸﾄﾌﾟﾚｯｼｬ連結中
      ANI     M7125  ; D70=003Ymin<PL-Yh-曲げ周長
      ORB
      ANB
      OUT     M7013  ; D70=003ﾘﾄﾗｸﾄﾌﾟﾚｯｼｬ後退仮
      MRD
      AND     M7013  ; D70=003ﾘﾄﾗｸﾄﾌﾟﾚｯｼｬ後退仮
      AND     M7008  ; D70=003干渉確認用接点
      MOV     K4 D70
      MPP
      OUT     M7008  ; D70=003干渉確認用接点
      MPP
      AND=    D70 K4  ; 自動運転ｽﾃｯﾌﾟMAIN
      AND     M3  ; ｽﾃｯﾌﾟ歩進
      MOV     K5 D70
209   LD      SM400  ; 常時 ON
      MPS
      AND=    D70 K5  ; 自動運転ｽﾃｯﾌﾟMAIN
      MPS
      ANI     T201  ; ﾘﾄﾗｸﾄﾌﾟﾚｯｼｬ昇降下降端遅延
      OUT     M7108  ; D70=005ﾘﾄﾗｸﾄﾌﾟﾚｯｼｬ下降
      MPP
      AND     T201  ; ﾘﾄﾗｸﾄﾌﾟﾚｯｼｬ昇降下降端遅延
      MOV     K6 D70
      MPP
      AND=    D70 K6  ; 自動運転ｽﾃｯﾌﾟMAIN
      AND     M3  ; ｽﾃｯﾌﾟ歩進
      MPS
      AND     M361  ; 曲げﾘﾄﾗｸﾄﾌﾟﾚｯｼｬ必要
      MOV     K8 D70
      MPP
      ANI     M361  ; 曲げﾘﾄﾗｸﾄﾌﾟﾚｯｼｬ必要
      MOV     K13 D70
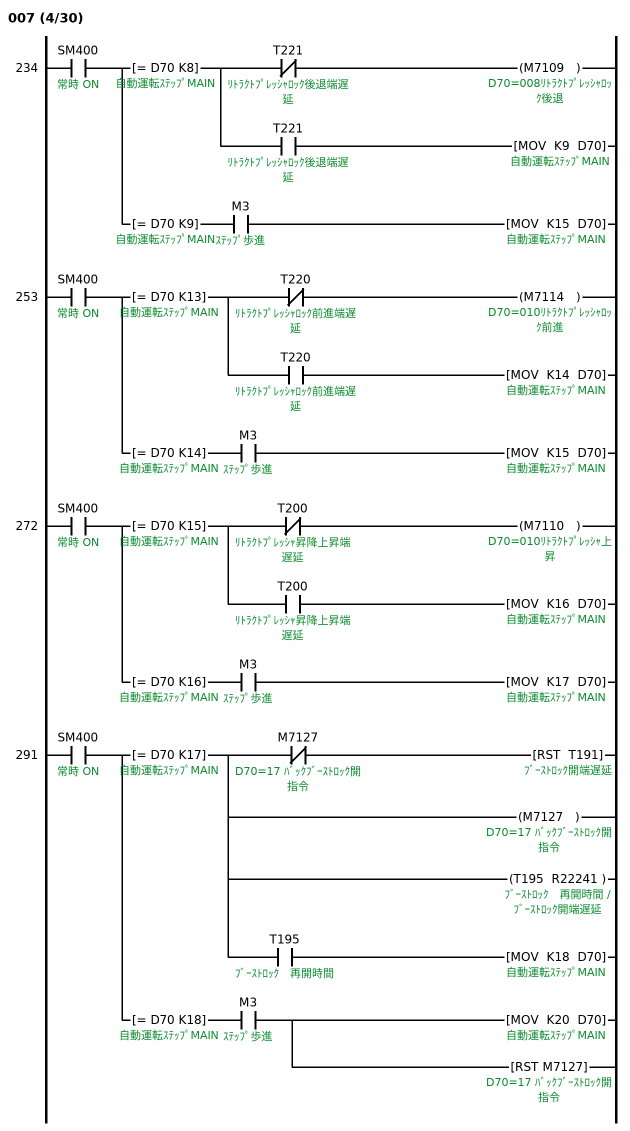
234   LD      SM400  ; 常時 ON
      MPS
      AND=    D70 K8  ; 自動運転ｽﾃｯﾌﾟMAIN
      MPS
      ANI     T221  ; ﾘﾄﾗｸﾄﾌﾟﾚｯｼｬﾛｯｸ後退端遅延
      OUT     M7109  ; D70=008ﾘﾄﾗｸﾄﾌﾟﾚｯｼｬﾛｯｸ後退
      MPP
      AND     T221  ; ﾘﾄﾗｸﾄﾌﾟﾚｯｼｬﾛｯｸ後退端遅延
      MOV     K9 D70
      MPP
      AND=    D70 K9  ; 自動運転ｽﾃｯﾌﾟMAIN
      AND     M3  ; ｽﾃｯﾌﾟ歩進
      MOV     K15 D70
253   LD      SM400  ; 常時 ON
      MPS
      AND=    D70 K13  ; 自動運転ｽﾃｯﾌﾟMAIN
      MPS
      ANI     T220  ; ﾘﾄﾗｸﾄﾌﾟﾚｯｼｬﾛｯｸ前進端遅延
      OUT     M7114  ; D70=010ﾘﾄﾗｸﾄﾌﾟﾚｯｼｬﾛｯｸ前進
      MPP
      AND     T220  ; ﾘﾄﾗｸﾄﾌﾟﾚｯｼｬﾛｯｸ前進端遅延
      MOV     K14 D70
      MPP
      AND=    D70 K14  ; 自動運転ｽﾃｯﾌﾟMAIN
      AND     M3  ; ｽﾃｯﾌﾟ歩進
      MOV     K15 D70
272   LD      SM400  ; 常時 ON
      MPS
      AND=    D70 K15  ; 自動運転ｽﾃｯﾌﾟMAIN
      MPS
      ANI     T200  ; ﾘﾄﾗｸﾄﾌﾟﾚｯｼｬ昇降上昇端遅延
      OUT     M7110  ; D70=010ﾘﾄﾗｸﾄﾌﾟﾚｯｼｬ上昇
      MPP
      AND     T200  ; ﾘﾄﾗｸﾄﾌﾟﾚｯｼｬ昇降上昇端遅延
      MOV     K16 D70
      MPP
      AND=    D70 K16  ; 自動運転ｽﾃｯﾌﾟMAIN
      AND     M3  ; ｽﾃｯﾌﾟ歩進
      MOV     K17 D70
291   LD      SM400  ; 常時 ON
      MPS
      AND=    D70 K17  ; 自動運転ｽﾃｯﾌﾟMAIN
      MPS
      ANI     M7127  ; D70=17 ﾊﾞｯｸﾌﾞｰｽﾄﾛｯｸ開指令
      RST     T191  ; ﾌﾞｰｽﾄﾛｯｸ開端遅延
      MPP
      OUT     M7127  ; D70=17 ﾊﾞｯｸﾌﾞｰｽﾄﾛｯｸ開指令
      OUT     T195 R22241  ; ﾌﾞｰｽﾄﾛｯｸ　再開時間 / ﾌﾞｰｽﾄﾛｯｸ開端遅延
      AND     T195  ; ﾌﾞｰｽﾄﾛｯｸ　再開時間
      MOV     K18 D70
      MPP
      AND=    D70 K18  ; 自動運転ｽﾃｯﾌﾟMAIN
      AND     M3  ; ｽﾃｯﾌﾟ歩進
      MOV     K20 D70
      RST     M7127  ; D70=17 ﾊﾞｯｸﾌﾞｰｽﾄﾛｯｸ開指令
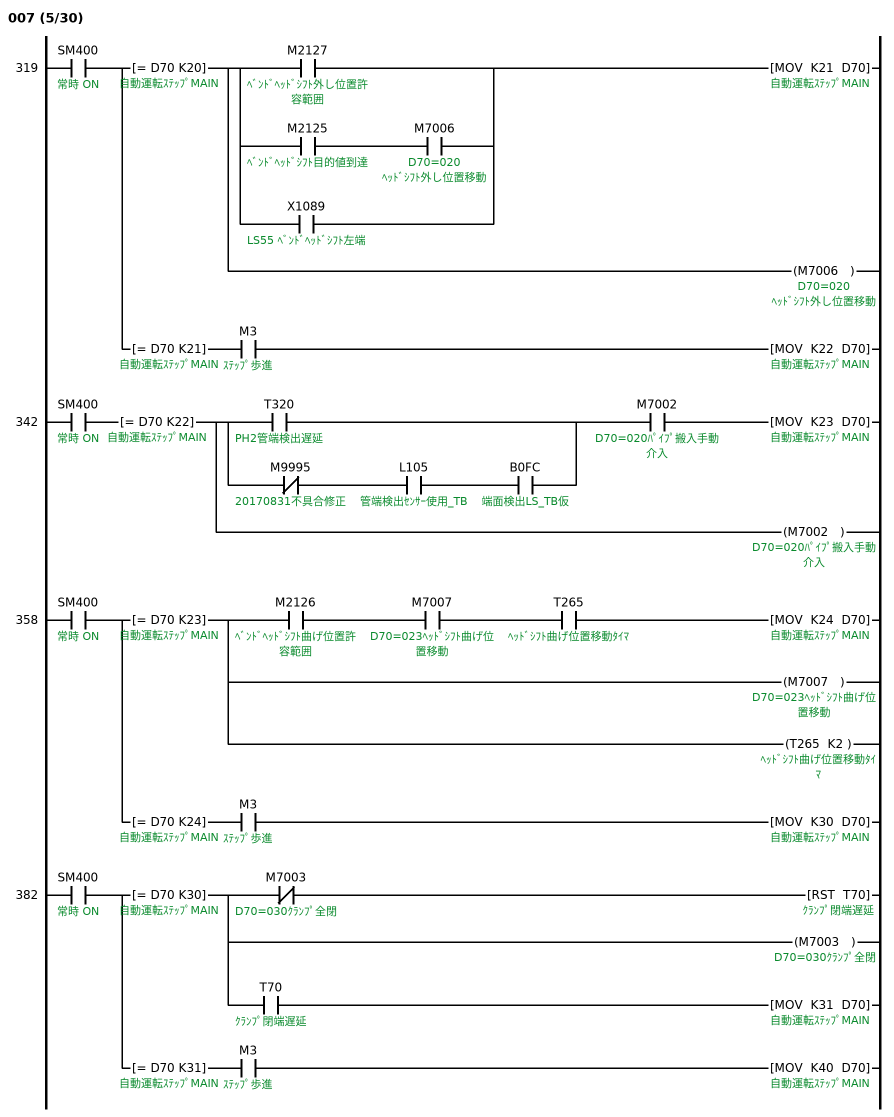
319   LD      SM400  ; 常時 ON
      MPS
      AND=    D70 K20  ; 自動運転ｽﾃｯﾌﾟMAIN
      MPS
      LD      M2127  ; ﾍﾞﾝﾄﾞﾍｯﾄﾞｼﾌﾄ外し位置許容範囲
      LD      M2125  ; ﾍﾞﾝﾄﾞﾍｯﾄﾞｼﾌﾄ目的値到達
      AND     M7006  ; D70=020 ﾍｯﾄﾞｼﾌﾄ外し位置移動
      ORB
      OR      X1089  ; LS55 ﾍﾞﾝﾄﾞﾍｯﾄﾞｼﾌﾄ左端
      ANB
      MOV     K21 D70
      MPP
      OUT     M7006  ; D70=020 ﾍｯﾄﾞｼﾌﾄ外し位置移動
      MPP
      AND=    D70 K21  ; 自動運転ｽﾃｯﾌﾟMAIN
      AND     M3  ; ｽﾃｯﾌﾟ歩進
      MOV     K22 D70
342   LD      SM400  ; 常時 ON
      AND=    D70 K22  ; 自動運転ｽﾃｯﾌﾟMAIN
      MPS
      LD      T320  ; PH2管端検出遅延
      LDI     M9995  ; 20170831不具合修正
      AND     L105  ; 管端検出ｾﾝｻｰ使用_TB
      AND     B0FC  ; 端面検出LS_TB仮
      ORB
      ANB
      AND     M7002  ; D70=020ﾊﾟｲﾌﾟ搬入手動介入
      MOV     K23 D70
      MPP
      OUT     M7002  ; D70=020ﾊﾟｲﾌﾟ搬入手動介入
358   LD      SM400  ; 常時 ON
      MPS
      AND=    D70 K23  ; 自動運転ｽﾃｯﾌﾟMAIN
      MPS
      AND     M2126  ; ﾍﾞﾝﾄﾞﾍｯﾄﾞｼﾌﾄ曲げ位置許容範囲
      AND     M7007  ; D70=023ﾍｯﾄﾞｼﾌﾄ曲げ位置移動
      AND     T265  ; ﾍｯﾄﾞｼﾌﾄ曲げ位置移動ﾀｲﾏ
      MOV     K24 D70
      MPP
      OUT     M7007  ; D70=023ﾍｯﾄﾞｼﾌﾄ曲げ位置移動
      OUT     T265 K2  ; ﾍｯﾄﾞｼﾌﾄ曲げ位置移動ﾀｲﾏ
      MPP
      AND=    D70 K24  ; 自動運転ｽﾃｯﾌﾟMAIN
      AND     M3  ; ｽﾃｯﾌﾟ歩進
      MOV     K30 D70
382   LD      SM400  ; 常時 ON
      MPS
      AND=    D70 K30  ; 自動運転ｽﾃｯﾌﾟMAIN
      MPS
      ANI     M7003  ; D70=030ｸﾗﾝﾌﾟ全閉
      RST     T70  ; ｸﾗﾝﾌﾟ閉端遅延
      MPP
      OUT     M7003  ; D70=030ｸﾗﾝﾌﾟ全閉
      AND     T70  ; ｸﾗﾝﾌﾟ閉端遅延
      MOV     K31 D70
      MPP
      AND=    D70 K31  ; 自動運転ｽﾃｯﾌﾟMAIN
      AND     M3  ; ｽﾃｯﾌﾟ歩進
      MOV     K40 D70
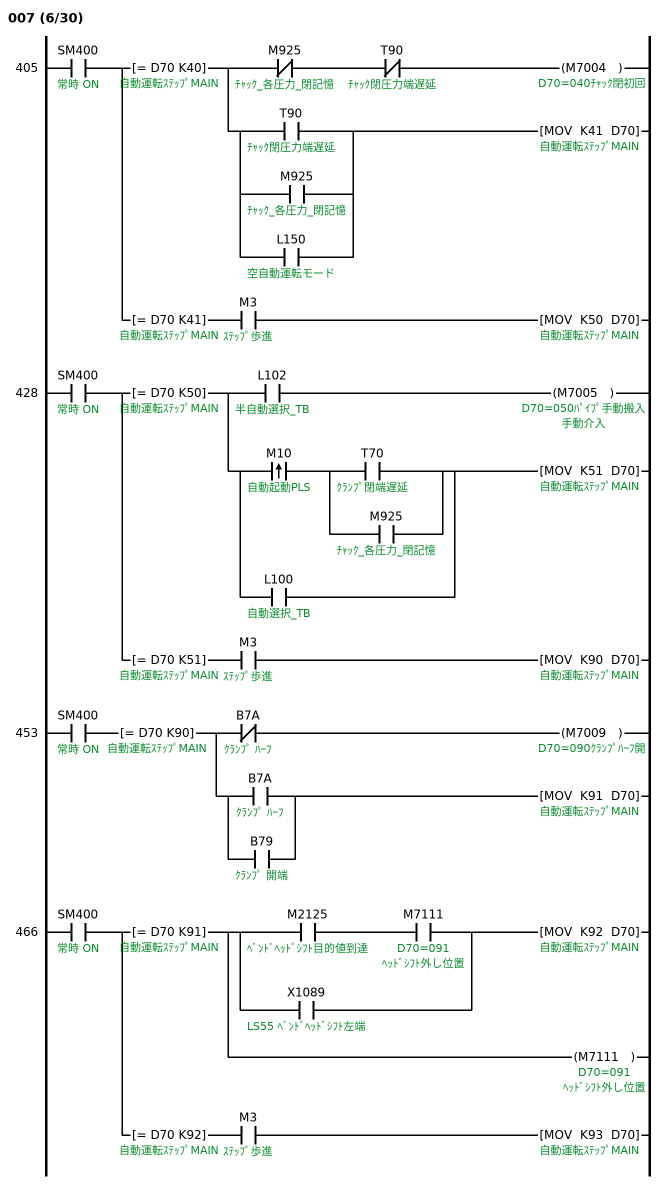
405   LD      SM400  ; 常時 ON
      MPS
      AND=    D70 K40  ; 自動運転ｽﾃｯﾌﾟMAIN
      MPS
      ANI     M925  ; ﾁｬｯｸ_各圧力_閉記憶
      ANI     T90  ; ﾁｬｯｸ閉圧力端遅延
      OUT     M7004  ; D70=040ﾁｬｯｸ閉初回
      MPP
      LD      T90  ; ﾁｬｯｸ閉圧力端遅延
      OR      M925  ; ﾁｬｯｸ_各圧力_閉記憶
      OR      L150  ; 空自動運転モード
      ANB
      MOV     K41 D70
      MPP
      AND=    D70 K41  ; 自動運転ｽﾃｯﾌﾟMAIN
      AND     M3  ; ｽﾃｯﾌﾟ歩進
      MOV     K50 D70
428   LD      SM400  ; 常時 ON
      MPS
      AND=    D70 K50  ; 自動運転ｽﾃｯﾌﾟMAIN
      MPS
      AND     L102  ; 半自動選択_TB
      OUT     M7005  ; D70=050ﾊﾟｲﾌﾟ手動搬入手動介入
      MPP
      LDP     M10  ; 自動起動PLS
      LD      T70  ; ｸﾗﾝﾌﾟ閉端遅延
      OR      M925  ; ﾁｬｯｸ_各圧力_閉記憶
      ANB
      OR      L100  ; 自動選択_TB
      ANB
      MOV     K51 D70
      MPP
      AND=    D70 K51  ; 自動運転ｽﾃｯﾌﾟMAIN
      AND     M3  ; ｽﾃｯﾌﾟ歩進
      MOV     K90 D70
453   LD      SM400  ; 常時 ON
      AND=    D70 K90  ; 自動運転ｽﾃｯﾌﾟMAIN
      MPS
      ANI     B7A  ; ｸﾗﾝﾌﾟ ﾊｰﾌ
      OUT     M7009  ; D70=090ｸﾗﾝﾌﾟﾊｰﾌ開
      MPP
      LD      B7A  ; ｸﾗﾝﾌﾟ ﾊｰﾌ
      OR      B79  ; ｸﾗﾝﾌﾟ 開端
      ANB
      MOV     K91 D70
466   LD      SM400  ; 常時 ON
      MPS
      AND=    D70 K91  ; 自動運転ｽﾃｯﾌﾟMAIN
      MPS
      LD      M2125  ; ﾍﾞﾝﾄﾞﾍｯﾄﾞｼﾌﾄ目的値到達
      AND     M7111  ; D70=091 ﾍｯﾄﾞｼﾌﾄ外し位置
      OR      X1089  ; LS55 ﾍﾞﾝﾄﾞﾍｯﾄﾞｼﾌﾄ左端
      ANB
      MOV     K92 D70
      MPP
      OUT     M7111  ; D70=091 ﾍｯﾄﾞｼﾌﾄ外し位置
      MPP
      AND=    D70 K92  ; 自動運転ｽﾃｯﾌﾟMAIN
      AND     M3  ; ｽﾃｯﾌﾟ歩進
      MOV     K93 D70
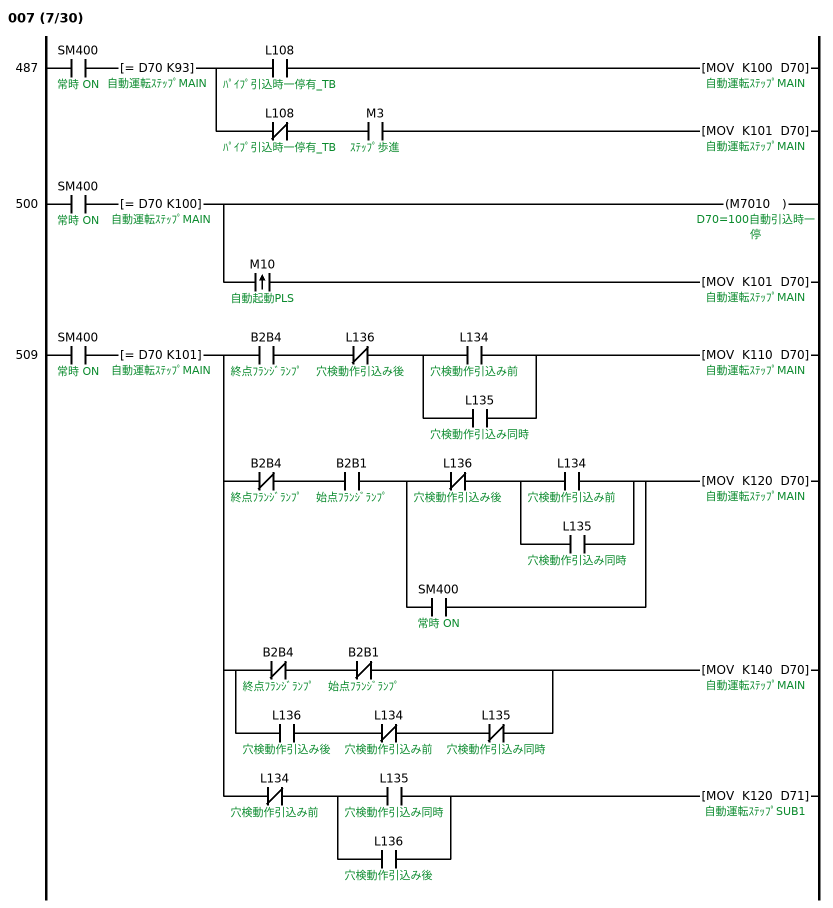
487   LD      SM400  ; 常時 ON
      AND=    D70 K93  ; 自動運転ｽﾃｯﾌﾟMAIN
      MPS
      AND     L108  ; ﾊﾟｲﾌﾟ引込時一停有_TB
      MOV     K100 D70
      MPP
      ANI     L108  ; ﾊﾟｲﾌﾟ引込時一停有_TB
      AND     M3  ; ｽﾃｯﾌﾟ歩進
      MOV     K101 D70
500   LD      SM400  ; 常時 ON
      AND=    D70 K100  ; 自動運転ｽﾃｯﾌﾟMAIN
      OUT     M7010  ; D70=100自動引込時一停
      ANDP    M10  ; 自動起動PLS
      MOV     K101 D70
509   LD      SM400  ; 常時 ON
      AND=    D70 K101  ; 自動運転ｽﾃｯﾌﾟMAIN
      MPS
      AND     B2B4  ; 終点ﾌﾗﾝｼﾞﾗﾝﾌﾟ
      ANI     L136  ; 穴検動作引込み後
      LD      L134  ; 穴検動作引込み前
      OR      L135  ; 穴検動作引込み同時
      ANB
      MOV     K110 D70
      MRD
      ANI     B2B4  ; 終点ﾌﾗﾝｼﾞﾗﾝﾌﾟ
      AND     B2B1  ; 始点ﾌﾗﾝｼﾞﾗﾝﾌﾟ
      LDI     L136  ; 穴検動作引込み後
      LD      L134  ; 穴検動作引込み前
      OR      L135  ; 穴検動作引込み同時
      ANB
      OR      SM400  ; 常時 ON
      ANB
      MOV     K120 D70
      MRD
      LDI     B2B4  ; 終点ﾌﾗﾝｼﾞﾗﾝﾌﾟ
      ANI     B2B1  ; 始点ﾌﾗﾝｼﾞﾗﾝﾌﾟ
      LD      L136  ; 穴検動作引込み後
      ANI     L134  ; 穴検動作引込み前
      ANI     L135  ; 穴検動作引込み同時
      ORB
      ANB
      MOV     K140 D70
      MPP
      ANI     L134  ; 穴検動作引込み前
      LD      L135  ; 穴検動作引込み同時
      OR      L136  ; 穴検動作引込み後
      ANB
      MOV     K120 D71  ; 自動運転ｽﾃｯﾌﾟSUB1
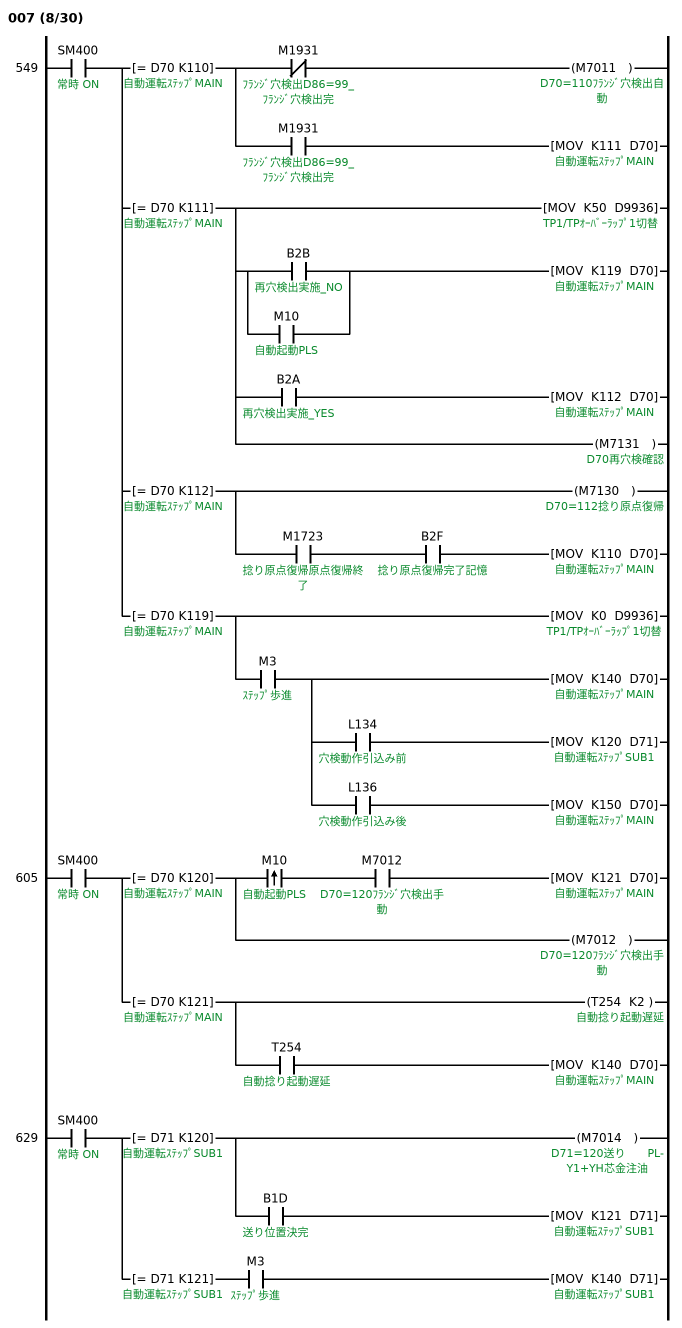
549   LD      SM400  ; 常時 ON
      MPS
      AND=    D70 K110  ; 自動運転ｽﾃｯﾌﾟMAIN
      MPS
      ANI     M1931  ; ﾌﾗﾝｼﾞ穴検出D86=99_ﾌﾗﾝｼﾞ穴検出完
      OUT     M7011  ; D70=110ﾌﾗﾝｼﾞ穴検出自動
      MPP
      AND     M1931  ; ﾌﾗﾝｼﾞ穴検出D86=99_ﾌﾗﾝｼﾞ穴検出完
      MOV     K111 D70
      MRD
      AND=    D70 K111  ; 自動運転ｽﾃｯﾌﾟMAIN
      MOV     K50 D9936  ; TP1/TPｵｰﾊﾞｰﾗｯﾌﾟ1切替
      MPS
      LD      B2B  ; 再穴検出実施_NO
      OR      M10  ; 自動起動PLS
      ANB
      MOV     K119 D70
      MRD
      AND     B2A  ; 再穴検出実施_YES
      MOV     K112 D70
      MPP
      OUT     M7131  ; D70再穴検確認
      MRD
      AND=    D70 K112  ; 自動運転ｽﾃｯﾌﾟMAIN
      OUT     M7130  ; D70=112捻り原点復帰
      AND     M1723  ; 捻り原点復帰原点復帰終了
      AND     B2F  ; 捻り原点復帰完了記憶
      MOV     K110 D70
      MPP
      AND=    D70 K119  ; 自動運転ｽﾃｯﾌﾟMAIN
      MOV     K0 D9936
      AND     M3  ; ｽﾃｯﾌﾟ歩進
      MOV     K140 D70
      MPS
      AND     L134  ; 穴検動作引込み前
      MOV     K120 D71
      MPP
      AND     L136  ; 穴検動作引込み後
      MOV     K150 D70
605   LD      SM400  ; 常時 ON
      MPS
      AND=    D70 K120  ; 自動運転ｽﾃｯﾌﾟMAIN
      MPS
      ANDP    M10  ; 自動起動PLS
      AND     M7012  ; D70=120ﾌﾗﾝｼﾞ穴検出手動
      MOV     K121 D70
      MPP
      OUT     M7012  ; D70=120ﾌﾗﾝｼﾞ穴検出手動
      MPP
      AND=    D70 K121  ; 自動運転ｽﾃｯﾌﾟMAIN
      OUT     T254 K2  ; 自動捻り起動遅延
      AND     T254  ; 自動捻り起動遅延
      MOV     K140 D70
629   LD      SM400  ; 常時 ON
      MPS
      AND=    D71 K120  ; 自動運転ｽﾃｯﾌﾟSUB1
      OUT     M7014  ; D71=120送り　　PL-Y1+YH芯金注油
      AND     B1D  ; 送り位置決完
      MOV     K121 D71
      MPP
      AND=    D71 K121  ; 自動運転ｽﾃｯﾌﾟSUB1
      AND     M3  ; ｽﾃｯﾌﾟ歩進
      MOV     K140 D71
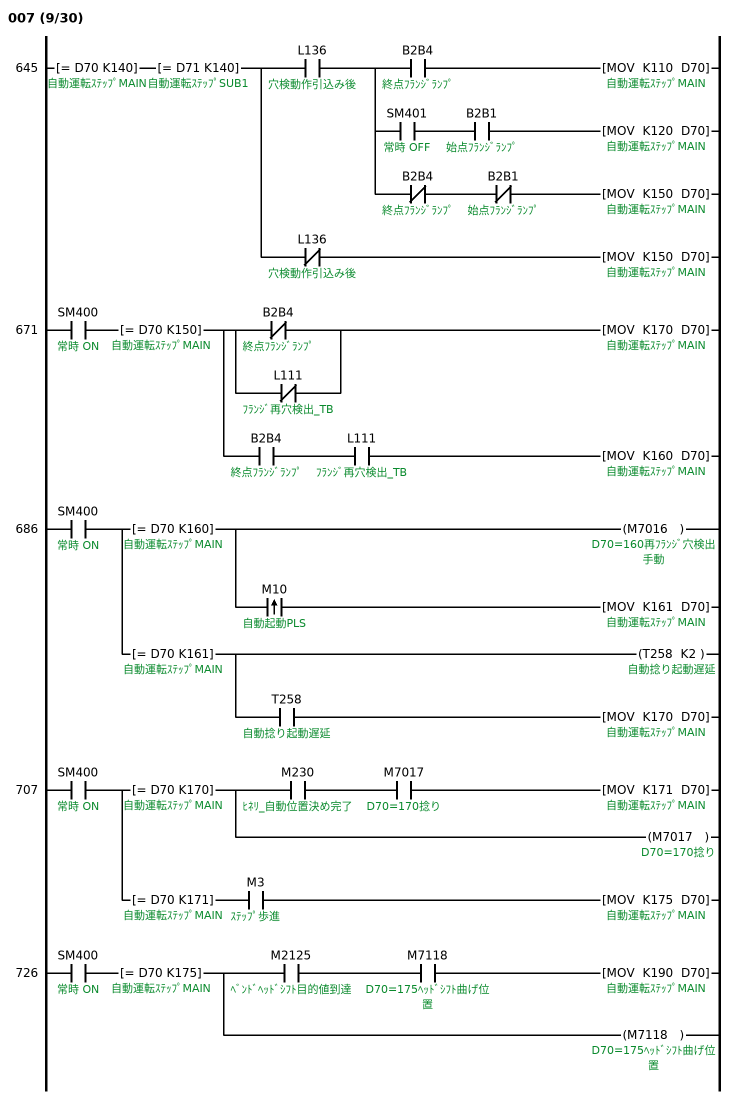
645   LD=     D70 K140  ; 自動運転ｽﾃｯﾌﾟMAIN
      AND=    D71 K140  ; 自動運転ｽﾃｯﾌﾟSUB1
      MPS
      AND     L136  ; 穴検動作引込み後
      MPS
      AND     B2B4  ; 終点ﾌﾗﾝｼﾞﾗﾝﾌﾟ
      MOV     K110 D70
      MRD
      AND     SM401  ; 常時 OFF
      AND     B2B1  ; 始点ﾌﾗﾝｼﾞﾗﾝﾌﾟ
      MOV     K120 D70
      MPP
      ANI     B2B4  ; 終点ﾌﾗﾝｼﾞﾗﾝﾌﾟ
      ANI     B2B1  ; 始点ﾌﾗﾝｼﾞﾗﾝﾌﾟ
      MOV     K150 D70
      MPP
      ANI     L136  ; 穴検動作引込み後
      MOV     K150 D70
671   LD      SM400  ; 常時 ON
      AND=    D70 K150  ; 自動運転ｽﾃｯﾌﾟMAIN
      MPS
      LDI     B2B4  ; 終点ﾌﾗﾝｼﾞﾗﾝﾌﾟ
      ORI     L111  ; ﾌﾗﾝｼﾞ再穴検出_TB
      ANB
      MOV     K170 D70
      MPP
      AND     B2B4  ; 終点ﾌﾗﾝｼﾞﾗﾝﾌﾟ
      AND     L111  ; ﾌﾗﾝｼﾞ再穴検出_TB
      MOV     K160 D70
686   LD      SM400  ; 常時 ON
      MPS
      AND=    D70 K160  ; 自動運転ｽﾃｯﾌﾟMAIN
      OUT     M7016  ; D70=160再ﾌﾗﾝｼﾞ穴検出手動
      ANDP    M10  ; 自動起動PLS
      MOV     K161 D70
      MPP
      AND=    D70 K161  ; 自動運転ｽﾃｯﾌﾟMAIN
      OUT     T258 K2  ; 自動捻り起動遅延
      AND     T258  ; 自動捻り起動遅延
      MOV     K170 D70
707   LD      SM400  ; 常時 ON
      MPS
      AND=    D70 K170  ; 自動運転ｽﾃｯﾌﾟMAIN
      MPS
      AND     M230  ; ﾋﾈﾘ_自動位置決め完了
      AND     M7017  ; D70=170捻り
      MOV     K171 D70
      MPP
      OUT     M7017  ; D70=170捻り
      MPP
      AND=    D70 K171  ; 自動運転ｽﾃｯﾌﾟMAIN
      AND     M3  ; ｽﾃｯﾌﾟ歩進
      MOV     K175 D70
726   LD      SM400  ; 常時 ON
      AND=    D70 K175  ; 自動運転ｽﾃｯﾌﾟMAIN
      MPS
      AND     M2125  ; ﾍﾞﾝﾄﾞﾍｯﾄﾞｼﾌﾄ目的値到達
      AND     M7118  ; D70=175ﾍｯﾄﾞｼﾌﾄ曲げ位置
      MOV     K190 D70
      MPP
      OUT     M7118  ; D70=175ﾍｯﾄﾞｼﾌﾄ曲げ位置
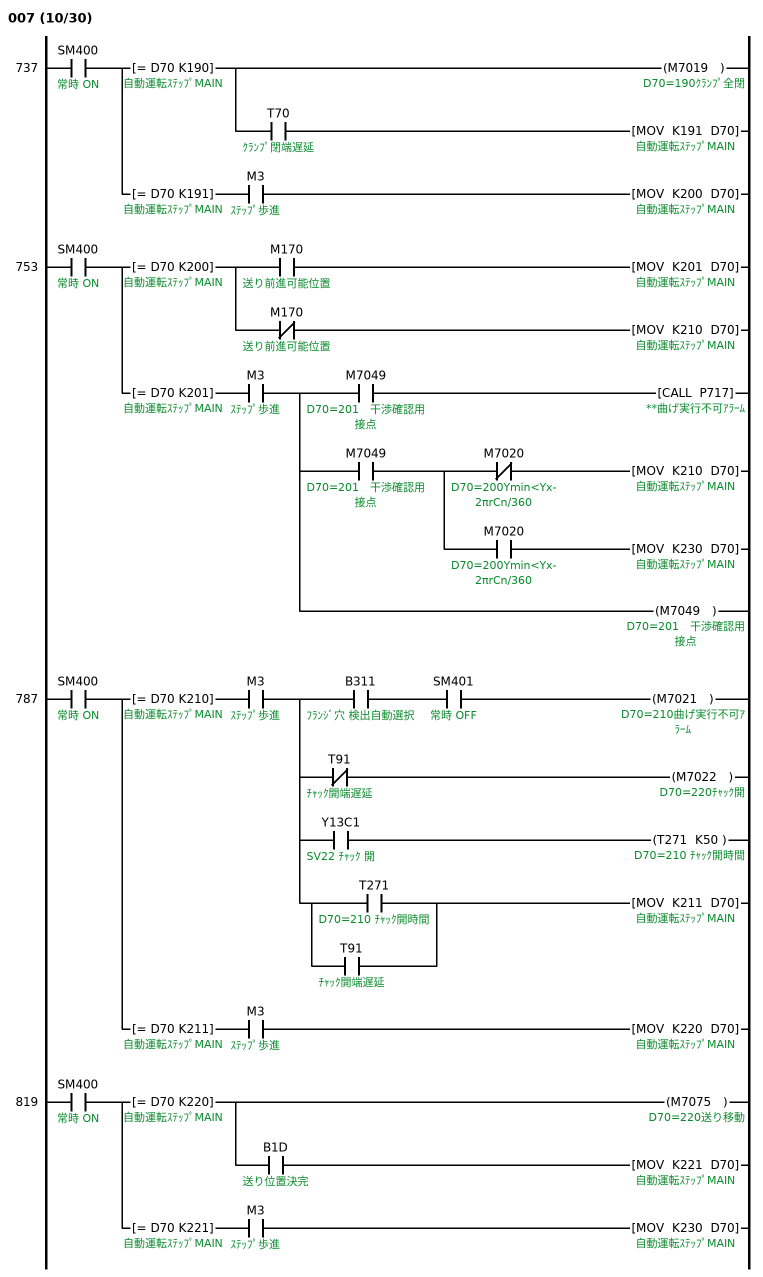
737   LD      SM400  ; 常時 ON
      MPS
      AND=    D70 K190  ; 自動運転ｽﾃｯﾌﾟMAIN
      OUT     M7019  ; D70=190ｸﾗﾝﾌﾟ全閉
      AND     T70  ; ｸﾗﾝﾌﾟ閉端遅延
      MOV     K191 D70
      MPP
      AND=    D70 K191  ; 自動運転ｽﾃｯﾌﾟMAIN
      AND     M3  ; ｽﾃｯﾌﾟ歩進
      MOV     K200 D70
753   LD      SM400  ; 常時 ON
      MPS
      AND=    D70 K200  ; 自動運転ｽﾃｯﾌﾟMAIN
      MPS
      AND     M170  ; 送り前進可能位置
      MOV     K201 D70
      MPP
      ANI     M170  ; 送り前進可能位置
      MOV     K210 D70
      MPP
      AND=    D70 K201  ; 自動運転ｽﾃｯﾌﾟMAIN
      AND     M3  ; ｽﾃｯﾌﾟ歩進
      MPS
      AND     M7049  ; D70=201　干渉確認用接点
      CALL    P717
      MRD
      AND     M7049  ; D70=201　干渉確認用接点
      MPS
      ANI     M7020  ; D70=200Ymin<Yx-2πrCn/360
      MOV     K210 D70
      MPP
      AND     M7020  ; D70=200Ymin<Yx-2πrCn/360
      MOV     K230 D70
      MPP
      OUT     M7049  ; D70=201　干渉確認用接点
787   LD      SM400  ; 常時 ON
      MPS
      AND=    D70 K210  ; 自動運転ｽﾃｯﾌﾟMAIN
      AND     M3  ; ｽﾃｯﾌﾟ歩進
      MPS
      AND     B311  ; ﾌﾗﾝｼﾞ穴 検出自動選択
      AND     SM401  ; 常時 OFF
      OUT     M7021  ; D70=210曲げ実行不可ｱﾗｰﾑ
      MRD
      ANI     T91  ; ﾁｬｯｸ開端遅延
      OUT     M7022  ; D70=220ﾁｬｯｸ開
      MRD
      AND     Y13C1  ; SV22 ﾁｬｯｸ 開
      OUT     T271 K50  ; D70=210 ﾁｬｯｸ開時間
      MPP
      LD      T271  ; D70=210 ﾁｬｯｸ開時間
      OR      T91  ; ﾁｬｯｸ開端遅延
      ANB
      MOV     K211 D70
      MPP
      AND=    D70 K211  ; 自動運転ｽﾃｯﾌﾟMAIN
      AND     M3  ; ｽﾃｯﾌﾟ歩進
      MOV     K220 D70
819   LD      SM400  ; 常時 ON
      MPS
      AND=    D70 K220  ; 自動運転ｽﾃｯﾌﾟMAIN
      OUT     M7075  ; D70=220送り移動
      AND     B1D  ; 送り位置決完
      MOV     K221 D70
      MPP
      AND=    D70 K221  ; 自動運転ｽﾃｯﾌﾟMAIN
      AND     M3  ; ｽﾃｯﾌﾟ歩進
      MOV     K230 D70
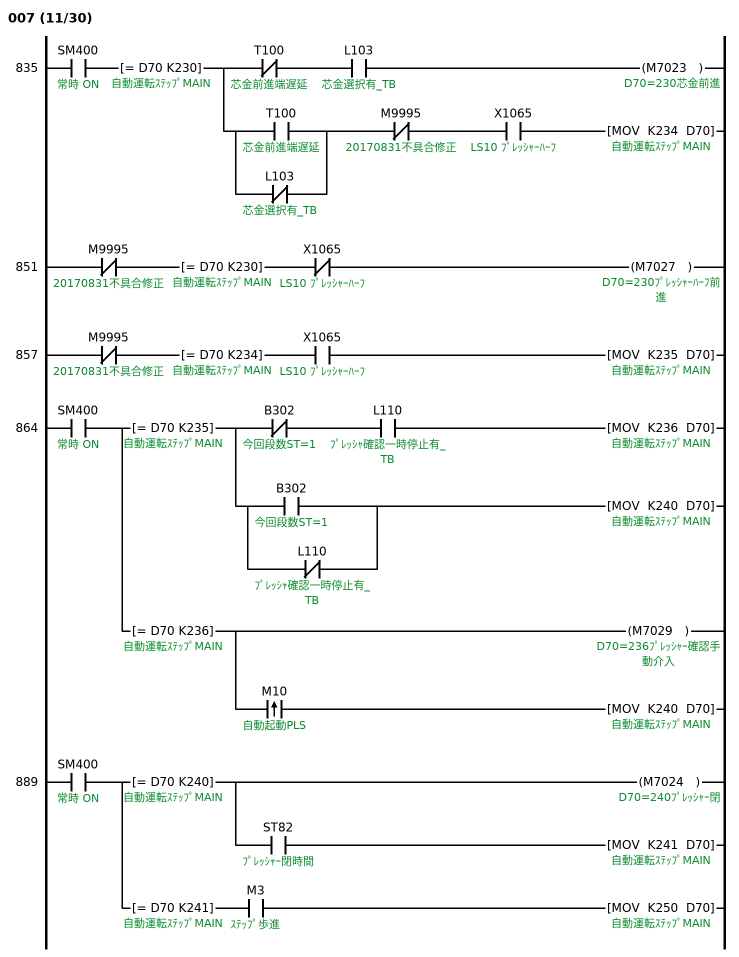
835   LD      SM400  ; 常時 ON
      AND=    D70 K230  ; 自動運転ｽﾃｯﾌﾟMAIN
      MPS
      ANI     T100  ; 芯金前進端遅延
      AND     L103  ; 芯金選択有_TB
      OUT     M7023  ; D70=230芯金前進
      MPP
      LD      T100  ; 芯金前進端遅延
      ORI     L103  ; 芯金選択有_TB
      ANB
      ANI     M9995  ; 20170831不具合修正
      AND     X1065  ; LS10 ﾌﾟﾚｯｼｬｰﾊｰﾌ
      MOV     K234 D70
851   LDI     M9995  ; 20170831不具合修正
      AND=    D70 K230  ; 自動運転ｽﾃｯﾌﾟMAIN
      ANI     X1065  ; LS10 ﾌﾟﾚｯｼｬｰﾊｰﾌ
      OUT     M7027  ; D70=230ﾌﾟﾚｯｼｬｰﾊｰﾌ前進
857   LDI     M9995  ; 20170831不具合修正
      AND=    D70 K234  ; 自動運転ｽﾃｯﾌﾟMAIN
      AND     X1065  ; LS10 ﾌﾟﾚｯｼｬｰﾊｰﾌ
      MOV     K235 D70
864   LD      SM400  ; 常時 ON
      MPS
      AND=    D70 K235  ; 自動運転ｽﾃｯﾌﾟMAIN
      MPS
      ANI     B302  ; 今回段数ST=1
      AND     L110  ; ﾌﾟﾚｯｼｬ確認一時停止有_TB
      MOV     K236 D70
      MPP
      LD      B302  ; 今回段数ST=1
      ORI     L110  ; ﾌﾟﾚｯｼｬ確認一時停止有_TB
      ANB
      MOV     K240 D70
      MPP
      AND=    D70 K236  ; 自動運転ｽﾃｯﾌﾟMAIN
      OUT     M7029  ; D70=236ﾌﾟﾚｯｼｬｰ確認手動介入
      ANDP    M10  ; 自動起動PLS
      MOV     K240 D70
889   LD      SM400  ; 常時 ON
      MPS
      AND=    D70 K240  ; 自動運転ｽﾃｯﾌﾟMAIN
      OUT     M7024  ; D70=240ﾌﾟﾚｯｼｬｰ閉
      AND     ST82  ; ﾌﾟﾚｯｼｬｰ閉時間
      MOV     K241 D70
      MPP
      AND=    D70 K241  ; 自動運転ｽﾃｯﾌﾟMAIN
      AND     M3  ; ｽﾃｯﾌﾟ歩進
      MOV     K250 D70
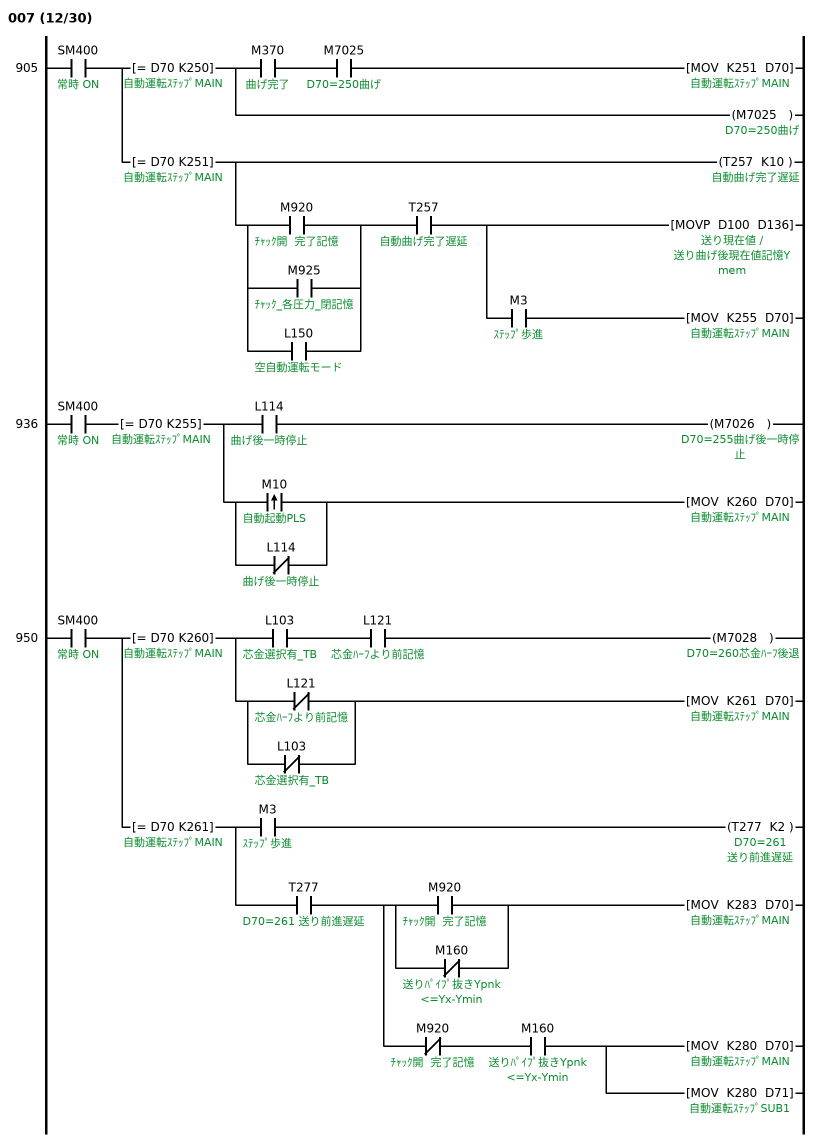
905   LD      SM400  ; 常時 ON
      MPS
      AND=    D70 K250  ; 自動運転ｽﾃｯﾌﾟMAIN
      MPS
      AND     M370  ; 曲げ完了
      AND     M7025  ; D70=250曲げ
      MOV     K251 D70
      MPP
      OUT     M7025  ; D70=250曲げ
      MPP
      AND=    D70 K251  ; 自動運転ｽﾃｯﾌﾟMAIN
      OUT     T257 K10  ; 自動曲げ完了遅延
      LD      M920  ; ﾁｬｯｸ開  完了記憶
      OR      M925  ; ﾁｬｯｸ_各圧力_閉記憶
      OR      L150  ; 空自動運転モード
      ANB
      AND     T257  ; 自動曲げ完了遅延
      MOVP    D100 D136  ; 送り現在値 / 送り曲げ後現在値記憶Ymem
      AND     M3  ; ｽﾃｯﾌﾟ歩進
      MOV     K255 D70
936   LD      SM400  ; 常時 ON
      AND=    D70 K255  ; 自動運転ｽﾃｯﾌﾟMAIN
      MPS
      AND     L114  ; 曲げ後一時停止
      OUT     M7026  ; D70=255曲げ後一時停止
      MPP
      LDP     M10  ; 自動起動PLS
      ORI     L114  ; 曲げ後一時停止
      ANB
      MOV     K260 D70
950   LD      SM400  ; 常時 ON
      MPS
      AND=    D70 K260  ; 自動運転ｽﾃｯﾌﾟMAIN
      MPS
      AND     L103  ; 芯金選択有_TB
      AND     L121  ; 芯金ﾊｰﾌより前記憶
      OUT     M7028  ; D70=260芯金ﾊｰﾌ後退
      MPP
      LDI     L121  ; 芯金ﾊｰﾌより前記憶
      ORI     L103  ; 芯金選択有_TB
      ANB
      MOV     K261 D70
      MPP
      AND=    D70 K261  ; 自動運転ｽﾃｯﾌﾟMAIN
      MPS
      AND     M3  ; ｽﾃｯﾌﾟ歩進
      OUT     T277 K2  ; D70=261 送り前進遅延
      MPP
      AND     T277  ; D70=261 送り前進遅延
      MPS
      LD      M920  ; ﾁｬｯｸ開  完了記憶
      ORI     M160  ; 送りﾊﾟｲﾌﾟ抜きYpnk <=Yx-Ymin
      ANB
      MOV     K283 D70
      MPP
      ANI     M920  ; ﾁｬｯｸ開  完了記憶
      AND     M160  ; 送りﾊﾟｲﾌﾟ抜きYpnk <=Yx-Ymin
      MOV     K280 D70
      MOV     K280 D71
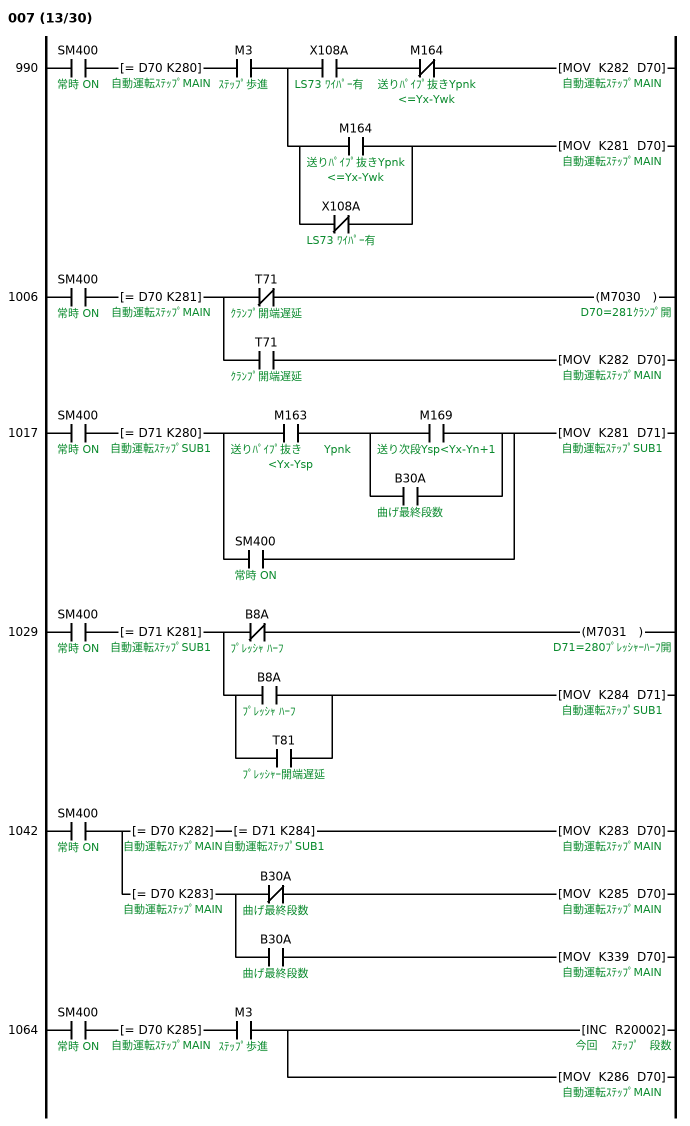
990   LD      SM400  ; 常時 ON
      AND=    D70 K280  ; 自動運転ｽﾃｯﾌﾟMAIN
      AND     M3  ; ｽﾃｯﾌﾟ歩進
      MPS
      AND     X108A  ; LS73 ﾜｲﾊﾟｰ有
      ANI     M164  ; 送りﾊﾟｲﾌﾟ抜きYpnk <=Yx-Ywk
      MOV     K282 D70
      MPP
      LD      M164  ; 送りﾊﾟｲﾌﾟ抜きYpnk <=Yx-Ywk
      ORI     X108A  ; LS73 ﾜｲﾊﾟｰ有
      ANB
      MOV     K281 D70
1006  LD      SM400  ; 常時 ON
      AND=    D70 K281  ; 自動運転ｽﾃｯﾌﾟMAIN
      MPS
      ANI     T71  ; ｸﾗﾝﾌﾟ開端遅延
      OUT     M7030  ; D70=281ｸﾗﾝﾌﾟ開
      MPP
      AND     T71  ; ｸﾗﾝﾌﾟ開端遅延
      MOV     K282 D70
1017  LD      SM400  ; 常時 ON
      AND=    D71 K280  ; 自動運転ｽﾃｯﾌﾟSUB1
      LD      M163  ; 送りﾊﾟｲﾌﾟ抜き　　Ypnk<Yx-Ysp
      LD      M169  ; 送り次段Ysp<Yx-Yn+1
      OR      B30A  ; 曲げ最終段数
      ANB
      OR      SM400  ; 常時 ON
      ANB
      MOV     K281 D71
1029  LD      SM400  ; 常時 ON
      AND=    D71 K281  ; 自動運転ｽﾃｯﾌﾟSUB1
      MPS
      ANI     B8A  ; ﾌﾟﾚｯｼｬ ﾊｰﾌ
      OUT     M7031  ; D71=280ﾌﾟﾚｯｼｬｰﾊｰﾌ開
      MPP
      LD      B8A  ; ﾌﾟﾚｯｼｬ ﾊｰﾌ
      OR      T81  ; ﾌﾟﾚｯｼｬｰ開端遅延
      ANB
      MOV     K284 D71
1042  LD      SM400  ; 常時 ON
      MPS
      AND=    D70 K282  ; 自動運転ｽﾃｯﾌﾟMAIN
      AND=    D71 K284  ; 自動運転ｽﾃｯﾌﾟSUB1
      MOV     K283 D70
      MPP
      AND=    D70 K283  ; 自動運転ｽﾃｯﾌﾟMAIN
      MPS
      ANI     B30A  ; 曲げ最終段数
      MOV     K285 D70
      MPP
      AND     B30A  ; 曲げ最終段数
      MOV     K339 D70
1064  LD      SM400  ; 常時 ON
      AND=    D70 K285  ; 自動運転ｽﾃｯﾌﾟMAIN
      AND     M3  ; ｽﾃｯﾌﾟ歩進
      INC     R20002
      MOV     K286 D70
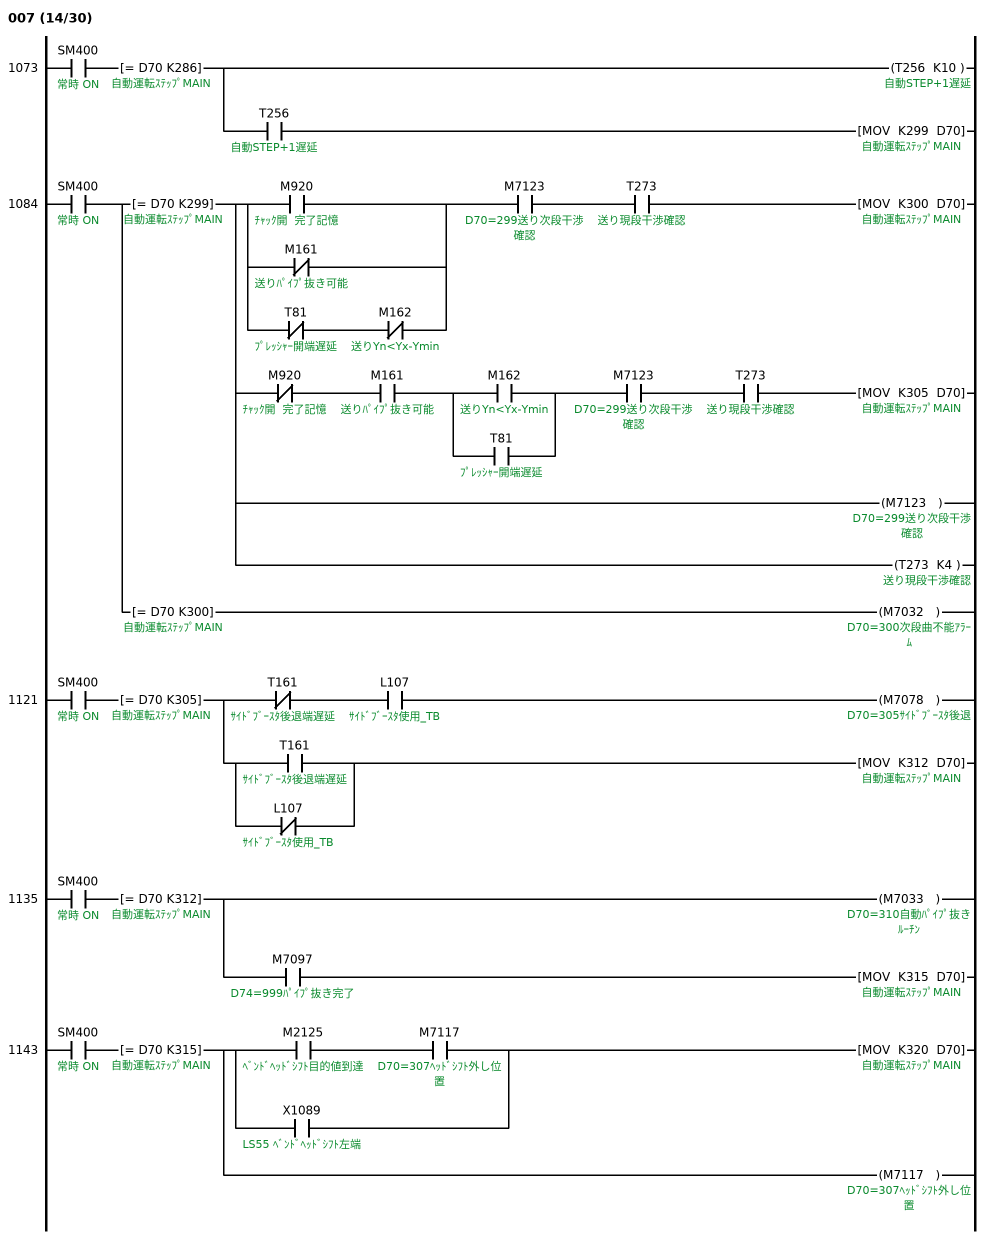
1073  LD      SM400  ; 常時 ON
      AND=    D70 K286  ; 自動運転ｽﾃｯﾌﾟMAIN
      OUT     T256 K10  ; 自動STEP+1遅延
      AND     T256  ; 自動STEP+1遅延
      MOV     K299 D70
1084  LD      SM400  ; 常時 ON
      MPS
      AND=    D70 K299  ; 自動運転ｽﾃｯﾌﾟMAIN
      MPS
      LD      M920  ; ﾁｬｯｸ開  完了記憶
      ORI     M161  ; 送りﾊﾟｲﾌﾟ抜き可能
      LDI     T81  ; ﾌﾟﾚｯｼｬｰ開端遅延
      ANI     M162  ; 送りYn<Yx-Ymin
      ORB
      ANB
      AND     M7123  ; D70=299送り次段干渉確認
      AND     T273  ; 送り現段干渉確認
      MOV     K300 D70
      MRD
      ANI     M920  ; ﾁｬｯｸ開  完了記憶
      AND     M161  ; 送りﾊﾟｲﾌﾟ抜き可能
      LD      M162  ; 送りYn<Yx-Ymin
      OR      T81  ; ﾌﾟﾚｯｼｬｰ開端遅延
      ANB
      AND     M7123  ; D70=299送り次段干渉確認
      AND     T273  ; 送り現段干渉確認
      MOV     K305 D70
      MPP
      OUT     M7123  ; D70=299送り次段干渉確認
      OUT     T273 K4  ; 送り現段干渉確認
      MPP
      AND=    D70 K300  ; 自動運転ｽﾃｯﾌﾟMAIN
      OUT     M7032  ; D70=300次段曲不能ｱﾗｰﾑ
1121  LD      SM400  ; 常時 ON
      AND=    D70 K305  ; 自動運転ｽﾃｯﾌﾟMAIN
      MPS
      ANI     T161  ; ｻｲﾄﾞﾌﾞｰｽﾀ後退端遅延
      AND     L107  ; ｻｲﾄﾞﾌﾞｰｽﾀ使用_TB
      OUT     M7078  ; D70=305ｻｲﾄﾞﾌﾞｰｽﾀ後退
      MPP
      LD      T161  ; ｻｲﾄﾞﾌﾞｰｽﾀ後退端遅延
      ORI     L107  ; ｻｲﾄﾞﾌﾞｰｽﾀ使用_TB
      ANB
      MOV     K312 D70
1135  LD      SM400  ; 常時 ON
      AND=    D70 K312  ; 自動運転ｽﾃｯﾌﾟMAIN
      OUT     M7033  ; D70=310自動ﾊﾟｲﾌﾟ抜きﾙｰﾁﾝ
      AND     M7097  ; D74=999ﾊﾟｲﾌﾟ抜き完了
      MOV     K315 D70
1143  LD      SM400  ; 常時 ON
      AND=    D70 K315  ; 自動運転ｽﾃｯﾌﾟMAIN
      MPS
      LD      M2125  ; ﾍﾞﾝﾄﾞﾍｯﾄﾞｼﾌﾄ目的値到達
      AND     M7117  ; D70=307ﾍｯﾄﾞｼﾌﾄ外し位置
      OR      X1089  ; LS55 ﾍﾞﾝﾄﾞﾍｯﾄﾞｼﾌﾄ左端
      ANB
      MOV     K320 D70
      MPP
      OUT     M7117  ; D70=307ﾍｯﾄﾞｼﾌﾄ外し位置
